   // GBK_TO_UNICODE[1865] := 16#547E;
   // GBK_TO_UNICODE[1866] := 16#85ED;
   // GBK_TO_UNICODE[1867] := 16#547F;
   // GBK_TO_UNICODE[1868] := 16#85EE;
   // GBK_TO_UNICODE[1869] := 16#5481;
   // GBK_TO_UNICODE[1870] := 16#85EF;
   // GBK_TO_UNICODE[1871] := 16#5483;
   // GBK_TO_UNICODE[1872] := 16#85F0;
   // GBK_TO_UNICODE[1873] := 16#5485;
   // GBK_TO_UNICODE[1874] := 16#85F1;
   // GBK_TO_UNICODE[1875] := 16#5487;
   // GBK_TO_UNICODE[1876] := 16#85F2;
   // GBK_TO_UNICODE[1877] := 16#5488;
   // GBK_TO_UNICODE[1878] := 16#85F3;
   // GBK_TO_UNICODE[1879] := 16#5489;
   // GBK_TO_UNICODE[1880] := 16#85F4;
   // GBK_TO_UNICODE[1881] := 16#548A;
   // GBK_TO_UNICODE[1882] := 16#85F5;
   // GBK_TO_UNICODE[1883] := 16#548D;
   // GBK_TO_UNICODE[1884] := 16#85F6;
   // GBK_TO_UNICODE[1885] := 16#5491;
   // GBK_TO_UNICODE[1886] := 16#85F7;
   // GBK_TO_UNICODE[1887] := 16#5493;
   // GBK_TO_UNICODE[1888] := 16#85F8;
   // GBK_TO_UNICODE[1889] := 16#5497;
   // GBK_TO_UNICODE[1890] := 16#85F9;
   // GBK_TO_UNICODE[1891] := 16#5498;
   // GBK_TO_UNICODE[1892] := 16#85FA;
   // GBK_TO_UNICODE[1893] := 16#549C;
   // GBK_TO_UNICODE[1894] := 16#85FB;
   // GBK_TO_UNICODE[1895] := 16#549E;
   // GBK_TO_UNICODE[1896] := 16#85FC;
   // GBK_TO_UNICODE[1897] := 16#549F;
   // GBK_TO_UNICODE[1898] := 16#85FD;
   // GBK_TO_UNICODE[1899] := 16#54A0;
   // GBK_TO_UNICODE[1900] := 16#85FE;
   // GBK_TO_UNICODE[1901] := 16#54A1;
   // GBK_TO_UNICODE[1902] := 16#8640;
   // GBK_TO_UNICODE[1903] := 16#54A2;
   // GBK_TO_UNICODE[1904] := 16#8641;
   // GBK_TO_UNICODE[1905] := 16#54A5;
   // GBK_TO_UNICODE[1906] := 16#8642;
   // GBK_TO_UNICODE[1907] := 16#54AE;
   // GBK_TO_UNICODE[1908] := 16#8643;
   // GBK_TO_UNICODE[1909] := 16#54B0;
   // GBK_TO_UNICODE[1910] := 16#8644;
   // GBK_TO_UNICODE[1911] := 16#54B2;
   // GBK_TO_UNICODE[1912] := 16#8645;
   // GBK_TO_UNICODE[1913] := 16#54B5;
   // GBK_TO_UNICODE[1914] := 16#8646;
   // GBK_TO_UNICODE[1915] := 16#54B6;
   // GBK_TO_UNICODE[1916] := 16#8647;
   // GBK_TO_UNICODE[1917] := 16#54B7;
   // GBK_TO_UNICODE[1918] := 16#8648;
   // GBK_TO_UNICODE[1919] := 16#54B9;
   // GBK_TO_UNICODE[1920] := 16#8649;
   // GBK_TO_UNICODE[1921] := 16#54BA;
   // GBK_TO_UNICODE[1922] := 16#864A;
   // GBK_TO_UNICODE[1923] := 16#54BC;
   // GBK_TO_UNICODE[1924] := 16#864B;
   // GBK_TO_UNICODE[1925] := 16#54BE;
   // GBK_TO_UNICODE[1926] := 16#864C;
   // GBK_TO_UNICODE[1927] := 16#54C3;
   // GBK_TO_UNICODE[1928] := 16#864D;
   // GBK_TO_UNICODE[1929] := 16#54C5;
   // GBK_TO_UNICODE[1930] := 16#864E;
   // GBK_TO_UNICODE[1931] := 16#54CA;
   // GBK_TO_UNICODE[1932] := 16#864F;
   // GBK_TO_UNICODE[1933] := 16#54CB;
   // GBK_TO_UNICODE[1934] := 16#8650;
   // GBK_TO_UNICODE[1935] := 16#54D6;
   // GBK_TO_UNICODE[1936] := 16#8651;
   // GBK_TO_UNICODE[1937] := 16#54D8;
   // GBK_TO_UNICODE[1938] := 16#8652;
   // GBK_TO_UNICODE[1939] := 16#54DB;
   // GBK_TO_UNICODE[1940] := 16#8653;
   // GBK_TO_UNICODE[1941] := 16#54E0;
   // GBK_TO_UNICODE[1942] := 16#8654;
   // GBK_TO_UNICODE[1943] := 16#54E1;
   // GBK_TO_UNICODE[1944] := 16#8655;
   // GBK_TO_UNICODE[1945] := 16#54E2;
   // GBK_TO_UNICODE[1946] := 16#8656;
   // GBK_TO_UNICODE[1947] := 16#54E3;
   // GBK_TO_UNICODE[1948] := 16#8657;
   // GBK_TO_UNICODE[1949] := 16#54E4;
   // GBK_TO_UNICODE[1950] := 16#8658;
   // GBK_TO_UNICODE[1951] := 16#54EB;
   // GBK_TO_UNICODE[1952] := 16#8659;
   // GBK_TO_UNICODE[1953] := 16#54EC;
   // GBK_TO_UNICODE[1954] := 16#865A;
   // GBK_TO_UNICODE[1955] := 16#54EF;
   // GBK_TO_UNICODE[1956] := 16#865B;
   // GBK_TO_UNICODE[1957] := 16#54F0;
   // GBK_TO_UNICODE[1958] := 16#865C;
   // GBK_TO_UNICODE[1959] := 16#54F1;
   // GBK_TO_UNICODE[1960] := 16#865D;
   // GBK_TO_UNICODE[1961] := 16#54F4;
   // GBK_TO_UNICODE[1962] := 16#865E;
   // GBK_TO_UNICODE[1963] := 16#54F5;
   // GBK_TO_UNICODE[1964] := 16#865F;
   // GBK_TO_UNICODE[1965] := 16#54F6;
   // GBK_TO_UNICODE[1966] := 16#8660;
   // GBK_TO_UNICODE[1967] := 16#54F7;
   // GBK_TO_UNICODE[1968] := 16#8661;
   // GBK_TO_UNICODE[1969] := 16#54F8;
   // GBK_TO_UNICODE[1970] := 16#8662;
   // GBK_TO_UNICODE[1971] := 16#54F9;
   // GBK_TO_UNICODE[1972] := 16#8663;
   // GBK_TO_UNICODE[1973] := 16#54FB;
   // GBK_TO_UNICODE[1974] := 16#8664;
   // GBK_TO_UNICODE[1975] := 16#54FE;
   // GBK_TO_UNICODE[1976] := 16#8665;
   // GBK_TO_UNICODE[1977] := 16#5500;
   // GBK_TO_UNICODE[1978] := 16#8666;
   // GBK_TO_UNICODE[1979] := 16#5502;
   // GBK_TO_UNICODE[1980] := 16#8667;
   // GBK_TO_UNICODE[1981] := 16#5503;
   // GBK_TO_UNICODE[1982] := 16#8668;
   // GBK_TO_UNICODE[1983] := 16#5504;
   // GBK_TO_UNICODE[1984] := 16#8669;
   // GBK_TO_UNICODE[1985] := 16#5505;
   // GBK_TO_UNICODE[1986] := 16#866A;
   // GBK_TO_UNICODE[1987] := 16#5508;
   // GBK_TO_UNICODE[1988] := 16#866B;
   // GBK_TO_UNICODE[1989] := 16#550A;
   // GBK_TO_UNICODE[1990] := 16#866C;
   // GBK_TO_UNICODE[1991] := 16#550B;
   // GBK_TO_UNICODE[1992] := 16#866D;
   // GBK_TO_UNICODE[1993] := 16#550C;
   // GBK_TO_UNICODE[1994] := 16#866E;
   // GBK_TO_UNICODE[1995] := 16#550D;
   // GBK_TO_UNICODE[1996] := 16#866F;
   // GBK_TO_UNICODE[1997] := 16#550E;
   // GBK_TO_UNICODE[1998] := 16#8670;
   // GBK_TO_UNICODE[1999] := 16#5512;
   // GBK_TO_UNICODE[2000] := 16#8671;
   // GBK_TO_UNICODE[2001] := 16#5513;
   // GBK_TO_UNICODE[2002] := 16#8672;
   // GBK_TO_UNICODE[2003] := 16#5515;
   // GBK_TO_UNICODE[2004] := 16#8673;
   // GBK_TO_UNICODE[2005] := 16#5516;
   // GBK_TO_UNICODE[2006] := 16#8674;
   // GBK_TO_UNICODE[2007] := 16#5517;
   // GBK_TO_UNICODE[2008] := 16#8675;
   // GBK_TO_UNICODE[2009] := 16#5518;
   // GBK_TO_UNICODE[2010] := 16#8676;
   // GBK_TO_UNICODE[2011] := 16#5519;
   // GBK_TO_UNICODE[2012] := 16#8677;
   // GBK_TO_UNICODE[2013] := 16#551A;
   // GBK_TO_UNICODE[2014] := 16#8678;
   // GBK_TO_UNICODE[2015] := 16#551C;
   // GBK_TO_UNICODE[2016] := 16#8679;
   // GBK_TO_UNICODE[2017] := 16#551D;
   // GBK_TO_UNICODE[2018] := 16#867A;
   // GBK_TO_UNICODE[2019] := 16#551E;
   // GBK_TO_UNICODE[2020] := 16#867B;
   // GBK_TO_UNICODE[2021] := 16#551F;
   // GBK_TO_UNICODE[2022] := 16#867C;
   // GBK_TO_UNICODE[2023] := 16#5521;
   // GBK_TO_UNICODE[2024] := 16#867D;
   // GBK_TO_UNICODE[2025] := 16#5525;
   // GBK_TO_UNICODE[2026] := 16#867E;
   // GBK_TO_UNICODE[2027] := 16#5526;
   // GBK_TO_UNICODE[2028] := 16#8680;
   // GBK_TO_UNICODE[2029] := 16#5528;
   // GBK_TO_UNICODE[2030] := 16#8681;
   // GBK_TO_UNICODE[2031] := 16#5529;
   // GBK_TO_UNICODE[2032] := 16#8682;
   // GBK_TO_UNICODE[2033] := 16#552B;
   // GBK_TO_UNICODE[2034] := 16#8683;
   // GBK_TO_UNICODE[2035] := 16#552D;
   // GBK_TO_UNICODE[2036] := 16#8684;
   // GBK_TO_UNICODE[2037] := 16#5532;
   // GBK_TO_UNICODE[2038] := 16#8685;
   // GBK_TO_UNICODE[2039] := 16#5534;
   // GBK_TO_UNICODE[2040] := 16#8686;
   // GBK_TO_UNICODE[2041] := 16#5535;
   // GBK_TO_UNICODE[2042] := 16#8687;
   // GBK_TO_UNICODE[2043] := 16#5536;
   // GBK_TO_UNICODE[2044] := 16#8688;
   // GBK_TO_UNICODE[2045] := 16#5538;
   // GBK_TO_UNICODE[2046] := 16#8689;
   // GBK_TO_UNICODE[2047] := 16#5539;
   // GBK_TO_UNICODE[2048] := 16#868A;
   // GBK_TO_UNICODE[2049] := 16#553A;
   // GBK_TO_UNICODE[2050] := 16#868B;
   // GBK_TO_UNICODE[2051] := 16#553B;
   // GBK_TO_UNICODE[2052] := 16#868C;
   // GBK_TO_UNICODE[2053] := 16#553D;
   // GBK_TO_UNICODE[2054] := 16#868D;
   // GBK_TO_UNICODE[2055] := 16#5540;
   // GBK_TO_UNICODE[2056] := 16#868E;
   // GBK_TO_UNICODE[2057] := 16#5542;
   // GBK_TO_UNICODE[2058] := 16#868F;
   // GBK_TO_UNICODE[2059] := 16#5545;
   // GBK_TO_UNICODE[2060] := 16#8690;
   // GBK_TO_UNICODE[2061] := 16#5547;
   // GBK_TO_UNICODE[2062] := 16#8691;
   // GBK_TO_UNICODE[2063] := 16#5548;
   // GBK_TO_UNICODE[2064] := 16#8692;
   // GBK_TO_UNICODE[2065] := 16#554B;
   // GBK_TO_UNICODE[2066] := 16#8693;
   // GBK_TO_UNICODE[2067] := 16#554C;
   // GBK_TO_UNICODE[2068] := 16#8694;
   // GBK_TO_UNICODE[2069] := 16#554D;
   // GBK_TO_UNICODE[2070] := 16#8695;
   // GBK_TO_UNICODE[2071] := 16#554E;
   // GBK_TO_UNICODE[2072] := 16#8696;
   // GBK_TO_UNICODE[2073] := 16#554F;
   // GBK_TO_UNICODE[2074] := 16#8697;
   // GBK_TO_UNICODE[2075] := 16#5551;
   // GBK_TO_UNICODE[2076] := 16#8698;
   // GBK_TO_UNICODE[2077] := 16#5552;
   // GBK_TO_UNICODE[2078] := 16#8699;
   // GBK_TO_UNICODE[2079] := 16#5553;
   // GBK_TO_UNICODE[2080] := 16#869A;
   // GBK_TO_UNICODE[2081] := 16#5554;
   // GBK_TO_UNICODE[2082] := 16#869B;
   // GBK_TO_UNICODE[2083] := 16#5557;
   // GBK_TO_UNICODE[2084] := 16#869C;
   // GBK_TO_UNICODE[2085] := 16#5558;
   // GBK_TO_UNICODE[2086] := 16#869D;
   // GBK_TO_UNICODE[2087] := 16#5559;
   // GBK_TO_UNICODE[2088] := 16#869E;
   // GBK_TO_UNICODE[2089] := 16#555A;
   // GBK_TO_UNICODE[2090] := 16#869F;
   // GBK_TO_UNICODE[2091] := 16#555B;
   // GBK_TO_UNICODE[2092] := 16#86A0;
   // GBK_TO_UNICODE[2093] := 16#555D;
   // GBK_TO_UNICODE[2094] := 16#86A1;
   // GBK_TO_UNICODE[2095] := 16#555E;
   // GBK_TO_UNICODE[2096] := 16#86A2;
   // GBK_TO_UNICODE[2097] := 16#555F;
   // GBK_TO_UNICODE[2098] := 16#86A3;
   // GBK_TO_UNICODE[2099] := 16#5560;
   // GBK_TO_UNICODE[2100] := 16#86A4;
   // GBK_TO_UNICODE[2101] := 16#5562;
   // GBK_TO_UNICODE[2102] := 16#86A5;
   // GBK_TO_UNICODE[2103] := 16#5563;
   // GBK_TO_UNICODE[2104] := 16#86A6;
   // GBK_TO_UNICODE[2105] := 16#5568;
   // GBK_TO_UNICODE[2106] := 16#86A7;
   // GBK_TO_UNICODE[2107] := 16#5569;
   // GBK_TO_UNICODE[2108] := 16#86A8;
   // GBK_TO_UNICODE[2109] := 16#556B;
   // GBK_TO_UNICODE[2110] := 16#86A9;
   // GBK_TO_UNICODE[2111] := 16#556F;
   // GBK_TO_UNICODE[2112] := 16#86AA;
   // GBK_TO_UNICODE[2113] := 16#5570;
   // GBK_TO_UNICODE[2114] := 16#86AB;
   // GBK_TO_UNICODE[2115] := 16#5571;
   // GBK_TO_UNICODE[2116] := 16#86AC;
   // GBK_TO_UNICODE[2117] := 16#5572;
   // GBK_TO_UNICODE[2118] := 16#86AD;
   // GBK_TO_UNICODE[2119] := 16#5573;
   // GBK_TO_UNICODE[2120] := 16#86AE;
   // GBK_TO_UNICODE[2121] := 16#5574;
   // GBK_TO_UNICODE[2122] := 16#86AF;
   // GBK_TO_UNICODE[2123] := 16#5579;
   // GBK_TO_UNICODE[2124] := 16#86B0;
   // GBK_TO_UNICODE[2125] := 16#557A;
   // GBK_TO_UNICODE[2126] := 16#86B1;
   // GBK_TO_UNICODE[2127] := 16#557D;
   // GBK_TO_UNICODE[2128] := 16#86B2;
   // GBK_TO_UNICODE[2129] := 16#557F;
   // GBK_TO_UNICODE[2130] := 16#86B3;
   // GBK_TO_UNICODE[2131] := 16#5585;
   // GBK_TO_UNICODE[2132] := 16#86B4;
   // GBK_TO_UNICODE[2133] := 16#5586;
   // GBK_TO_UNICODE[2134] := 16#86B5;
   // GBK_TO_UNICODE[2135] := 16#558C;
   // GBK_TO_UNICODE[2136] := 16#86B6;
   // GBK_TO_UNICODE[2137] := 16#558D;
   // GBK_TO_UNICODE[2138] := 16#86B7;
   // GBK_TO_UNICODE[2139] := 16#558E;
   // GBK_TO_UNICODE[2140] := 16#86B8;
   // GBK_TO_UNICODE[2141] := 16#5590;
   // GBK_TO_UNICODE[2142] := 16#86B9;
   // GBK_TO_UNICODE[2143] := 16#5592;
   // GBK_TO_UNICODE[2144] := 16#86BA;
   // GBK_TO_UNICODE[2145] := 16#5593;
   // GBK_TO_UNICODE[2146] := 16#86BB;
   // GBK_TO_UNICODE[2147] := 16#5595;
   // GBK_TO_UNICODE[2148] := 16#86BC;
   // GBK_TO_UNICODE[2149] := 16#5596;
   // GBK_TO_UNICODE[2150] := 16#86BD;
   // GBK_TO_UNICODE[2151] := 16#5597;
   // GBK_TO_UNICODE[2152] := 16#86BE;
   // GBK_TO_UNICODE[2153] := 16#559A;
   // GBK_TO_UNICODE[2154] := 16#86BF;
   // GBK_TO_UNICODE[2155] := 16#559B;
   // GBK_TO_UNICODE[2156] := 16#86C0;
   // GBK_TO_UNICODE[2157] := 16#559E;
   // GBK_TO_UNICODE[2158] := 16#86C1;
   // GBK_TO_UNICODE[2159] := 16#55A0;
   // GBK_TO_UNICODE[2160] := 16#86C2;
   // GBK_TO_UNICODE[2161] := 16#55A1;
   // GBK_TO_UNICODE[2162] := 16#86C3;
   // GBK_TO_UNICODE[2163] := 16#55A2;
   // GBK_TO_UNICODE[2164] := 16#86C4;
   // GBK_TO_UNICODE[2165] := 16#55A3;
   // GBK_TO_UNICODE[2166] := 16#86C5;
   // GBK_TO_UNICODE[2167] := 16#55A4;
   // GBK_TO_UNICODE[2168] := 16#86C6;
   // GBK_TO_UNICODE[2169] := 16#55A5;
   // GBK_TO_UNICODE[2170] := 16#86C7;
   // GBK_TO_UNICODE[2171] := 16#55A6;
   // GBK_TO_UNICODE[2172] := 16#86C8;
   // GBK_TO_UNICODE[2173] := 16#55A8;
   // GBK_TO_UNICODE[2174] := 16#86C9;
   // GBK_TO_UNICODE[2175] := 16#55A9;
   // GBK_TO_UNICODE[2176] := 16#86CA;
   // GBK_TO_UNICODE[2177] := 16#55AA;
   // GBK_TO_UNICODE[2178] := 16#86CB;
   // GBK_TO_UNICODE[2179] := 16#55AB;
   // GBK_TO_UNICODE[2180] := 16#86CC;
   // GBK_TO_UNICODE[2181] := 16#55AC;
   // GBK_TO_UNICODE[2182] := 16#86CD;
   // GBK_TO_UNICODE[2183] := 16#55AD;
   // GBK_TO_UNICODE[2184] := 16#86CE;
   // GBK_TO_UNICODE[2185] := 16#55AE;
   // GBK_TO_UNICODE[2186] := 16#86CF;
   // GBK_TO_UNICODE[2187] := 16#55AF;
   // GBK_TO_UNICODE[2188] := 16#86D0;
   // GBK_TO_UNICODE[2189] := 16#55B0;
   // GBK_TO_UNICODE[2190] := 16#86D1;
   // GBK_TO_UNICODE[2191] := 16#55B2;
   // GBK_TO_UNICODE[2192] := 16#86D2;
   // GBK_TO_UNICODE[2193] := 16#55B4;
   // GBK_TO_UNICODE[2194] := 16#86D3;
   // GBK_TO_UNICODE[2195] := 16#55B6;
   // GBK_TO_UNICODE[2196] := 16#86D4;
   // GBK_TO_UNICODE[2197] := 16#55B8;
   // GBK_TO_UNICODE[2198] := 16#86D5;
   // GBK_TO_UNICODE[2199] := 16#55BA;
   // GBK_TO_UNICODE[2200] := 16#86D6;
   // GBK_TO_UNICODE[2201] := 16#55BC;
   // GBK_TO_UNICODE[2202] := 16#86D7;
   // GBK_TO_UNICODE[2203] := 16#55BF;
   // GBK_TO_UNICODE[2204] := 16#86D8;
   // GBK_TO_UNICODE[2205] := 16#55C0;
   // GBK_TO_UNICODE[2206] := 16#86D9;
   // GBK_TO_UNICODE[2207] := 16#55C1;
   // GBK_TO_UNICODE[2208] := 16#86DA;
   // GBK_TO_UNICODE[2209] := 16#55C2;
   // GBK_TO_UNICODE[2210] := 16#86DB;
   // GBK_TO_UNICODE[2211] := 16#55C3;
   // GBK_TO_UNICODE[2212] := 16#86DC;
   // GBK_TO_UNICODE[2213] := 16#55C6;
   // GBK_TO_UNICODE[2214] := 16#86DD;
   // GBK_TO_UNICODE[2215] := 16#55C7;
   // GBK_TO_UNICODE[2216] := 16#86DE;
   // GBK_TO_UNICODE[2217] := 16#55C8;
   // GBK_TO_UNICODE[2218] := 16#86DF;
   // GBK_TO_UNICODE[2219] := 16#55CA;
   // GBK_TO_UNICODE[2220] := 16#86E0;
   // GBK_TO_UNICODE[2221] := 16#55CB;
   // GBK_TO_UNICODE[2222] := 16#86E1;
   // GBK_TO_UNICODE[2223] := 16#55CE;
   // GBK_TO_UNICODE[2224] := 16#86E2;
   // GBK_TO_UNICODE[2225] := 16#55CF;
   // GBK_TO_UNICODE[2226] := 16#86E3;
   // GBK_TO_UNICODE[2227] := 16#55D0;
   // GBK_TO_UNICODE[2228] := 16#86E4;
   // GBK_TO_UNICODE[2229] := 16#55D5;
   // GBK_TO_UNICODE[2230] := 16#86E5;
   // GBK_TO_UNICODE[2231] := 16#55D7;
   // GBK_TO_UNICODE[2232] := 16#86E6;
   // GBK_TO_UNICODE[2233] := 16#55D8;
   // GBK_TO_UNICODE[2234] := 16#86E7;
   // GBK_TO_UNICODE[2235] := 16#55D9;
   // GBK_TO_UNICODE[2236] := 16#86E8;
   // GBK_TO_UNICODE[2237] := 16#55DA;
   // GBK_TO_UNICODE[2238] := 16#86E9;
   // GBK_TO_UNICODE[2239] := 16#55DB;
   // GBK_TO_UNICODE[2240] := 16#86EA;
   // GBK_TO_UNICODE[2241] := 16#55DE;
   // GBK_TO_UNICODE[2242] := 16#86EB;
   // GBK_TO_UNICODE[2243] := 16#55E0;
   // GBK_TO_UNICODE[2244] := 16#86EC;
   // GBK_TO_UNICODE[2245] := 16#55E2;
   // GBK_TO_UNICODE[2246] := 16#86ED;
   // GBK_TO_UNICODE[2247] := 16#55E7;
   // GBK_TO_UNICODE[2248] := 16#86EE;
   // GBK_TO_UNICODE[2249] := 16#55E9;
   // GBK_TO_UNICODE[2250] := 16#86EF;
   // GBK_TO_UNICODE[2251] := 16#55ED;
   // GBK_TO_UNICODE[2252] := 16#86F0;
   // GBK_TO_UNICODE[2253] := 16#55EE;
   // GBK_TO_UNICODE[2254] := 16#86F1;
   // GBK_TO_UNICODE[2255] := 16#55F0;
   // GBK_TO_UNICODE[2256] := 16#86F2;
   // GBK_TO_UNICODE[2257] := 16#55F1;
   // GBK_TO_UNICODE[2258] := 16#86F3;
   // GBK_TO_UNICODE[2259] := 16#55F4;
   // GBK_TO_UNICODE[2260] := 16#86F4;
   // GBK_TO_UNICODE[2261] := 16#55F6;
   // GBK_TO_UNICODE[2262] := 16#86F5;
   // GBK_TO_UNICODE[2263] := 16#55F8;
   // GBK_TO_UNICODE[2264] := 16#86F6;
   // GBK_TO_UNICODE[2265] := 16#55F9;
   // GBK_TO_UNICODE[2266] := 16#86F7;
   // GBK_TO_UNICODE[2267] := 16#55FA;
   // GBK_TO_UNICODE[2268] := 16#86F8;
   // GBK_TO_UNICODE[2269] := 16#55FB;
   // GBK_TO_UNICODE[2270] := 16#86F9;
   // GBK_TO_UNICODE[2271] := 16#55FC;
   // GBK_TO_UNICODE[2272] := 16#86FA;
   // GBK_TO_UNICODE[2273] := 16#55FF;
   // GBK_TO_UNICODE[2274] := 16#86FB;
   // GBK_TO_UNICODE[2275] := 16#5602;
   // GBK_TO_UNICODE[2276] := 16#86FC;
   // GBK_TO_UNICODE[2277] := 16#5603;
   // GBK_TO_UNICODE[2278] := 16#86FD;
   // GBK_TO_UNICODE[2279] := 16#5604;
   // GBK_TO_UNICODE[2280] := 16#86FE;
   // GBK_TO_UNICODE[2281] := 16#5605;
   // GBK_TO_UNICODE[2282] := 16#8740;
   // GBK_TO_UNICODE[2283] := 16#5606;
   // GBK_TO_UNICODE[2284] := 16#8741;
   // GBK_TO_UNICODE[2285] := 16#5607;
   // GBK_TO_UNICODE[2286] := 16#8742;
   // GBK_TO_UNICODE[2287] := 16#560A;
   // GBK_TO_UNICODE[2288] := 16#8743;
   // GBK_TO_UNICODE[2289] := 16#560B;
   // GBK_TO_UNICODE[2290] := 16#8744;
   // GBK_TO_UNICODE[2291] := 16#560D;
   // GBK_TO_UNICODE[2292] := 16#8745;
   // GBK_TO_UNICODE[2293] := 16#5610;
   // GBK_TO_UNICODE[2294] := 16#8746;
   // GBK_TO_UNICODE[2295] := 16#5611;
   // GBK_TO_UNICODE[2296] := 16#8747;
   // GBK_TO_UNICODE[2297] := 16#5612;
   // GBK_TO_UNICODE[2298] := 16#8748;
   // GBK_TO_UNICODE[2299] := 16#5613;
   // GBK_TO_UNICODE[2300] := 16#8749;
   // GBK_TO_UNICODE[2301] := 16#5614;
   // GBK_TO_UNICODE[2302] := 16#874A;
   // GBK_TO_UNICODE[2303] := 16#5615;
   // GBK_TO_UNICODE[2304] := 16#874B;
   // GBK_TO_UNICODE[2305] := 16#5616;
   // GBK_TO_UNICODE[2306] := 16#874C;
   // GBK_TO_UNICODE[2307] := 16#5617;
   // GBK_TO_UNICODE[2308] := 16#874D;
   // GBK_TO_UNICODE[2309] := 16#5619;
   // GBK_TO_UNICODE[2310] := 16#874E;
   // GBK_TO_UNICODE[2311] := 16#561A;
   // GBK_TO_UNICODE[2312] := 16#874F;
   // GBK_TO_UNICODE[2313] := 16#561C;
   // GBK_TO_UNICODE[2314] := 16#8750;
   // GBK_TO_UNICODE[2315] := 16#561D;
   // GBK_TO_UNICODE[2316] := 16#8751;
   // GBK_TO_UNICODE[2317] := 16#5620;
   // GBK_TO_UNICODE[2318] := 16#8752;
   // GBK_TO_UNICODE[2319] := 16#5621;
   // GBK_TO_UNICODE[2320] := 16#8753;
   // GBK_TO_UNICODE[2321] := 16#5622;
   // GBK_TO_UNICODE[2322] := 16#8754;
   // GBK_TO_UNICODE[2323] := 16#5625;
   // GBK_TO_UNICODE[2324] := 16#8755;
   // GBK_TO_UNICODE[2325] := 16#5626;
   // GBK_TO_UNICODE[2326] := 16#8756;
   // GBK_TO_UNICODE[2327] := 16#5628;
   // GBK_TO_UNICODE[2328] := 16#8757;
   // GBK_TO_UNICODE[2329] := 16#5629;
   // GBK_TO_UNICODE[2330] := 16#8758;
   // GBK_TO_UNICODE[2331] := 16#562A;
   // GBK_TO_UNICODE[2332] := 16#8759;
   // GBK_TO_UNICODE[2333] := 16#562B;
   // GBK_TO_UNICODE[2334] := 16#875A;
   // GBK_TO_UNICODE[2335] := 16#562E;
   // GBK_TO_UNICODE[2336] := 16#875B;
   // GBK_TO_UNICODE[2337] := 16#562F;
   // GBK_TO_UNICODE[2338] := 16#875C;
   // GBK_TO_UNICODE[2339] := 16#5630;
   // GBK_TO_UNICODE[2340] := 16#875D;
   // GBK_TO_UNICODE[2341] := 16#5633;
   // GBK_TO_UNICODE[2342] := 16#875E;
   // GBK_TO_UNICODE[2343] := 16#5635;
   // GBK_TO_UNICODE[2344] := 16#875F;
   // GBK_TO_UNICODE[2345] := 16#5637;
   // GBK_TO_UNICODE[2346] := 16#8760;
   // GBK_TO_UNICODE[2347] := 16#5638;
   // GBK_TO_UNICODE[2348] := 16#8761;
   // GBK_TO_UNICODE[2349] := 16#563A;
   // GBK_TO_UNICODE[2350] := 16#8762;
   // GBK_TO_UNICODE[2351] := 16#563C;
   // GBK_TO_UNICODE[2352] := 16#8763;
   // GBK_TO_UNICODE[2353] := 16#563D;
   // GBK_TO_UNICODE[2354] := 16#8764;
   // GBK_TO_UNICODE[2355] := 16#563E;
   // GBK_TO_UNICODE[2356] := 16#8765;
   // GBK_TO_UNICODE[2357] := 16#5640;
   // GBK_TO_UNICODE[2358] := 16#8766;
   // GBK_TO_UNICODE[2359] := 16#5641;
   // GBK_TO_UNICODE[2360] := 16#8767;
   // GBK_TO_UNICODE[2361] := 16#5642;
   // GBK_TO_UNICODE[2362] := 16#8768;
   // GBK_TO_UNICODE[2363] := 16#5643;
   // GBK_TO_UNICODE[2364] := 16#8769;
   // GBK_TO_UNICODE[2365] := 16#5644;
   // GBK_TO_UNICODE[2366] := 16#876A;
   // GBK_TO_UNICODE[2367] := 16#5645;
   // GBK_TO_UNICODE[2368] := 16#876B;
   // GBK_TO_UNICODE[2369] := 16#5646;
   // GBK_TO_UNICODE[2370] := 16#876C;
   // GBK_TO_UNICODE[2371] := 16#5647;
   // GBK_TO_UNICODE[2372] := 16#876D;
   // GBK_TO_UNICODE[2373] := 16#5648;
   // GBK_TO_UNICODE[2374] := 16#876E;
   // GBK_TO_UNICODE[2375] := 16#5649;
   // GBK_TO_UNICODE[2376] := 16#876F;
   // GBK_TO_UNICODE[2377] := 16#564A;
   // GBK_TO_UNICODE[2378] := 16#8770;
   // GBK_TO_UNICODE[2379] := 16#564B;
   // GBK_TO_UNICODE[2380] := 16#8771;
   // GBK_TO_UNICODE[2381] := 16#564F;
   // GBK_TO_UNICODE[2382] := 16#8772;
   // GBK_TO_UNICODE[2383] := 16#5650;
   // GBK_TO_UNICODE[2384] := 16#8773;
   // GBK_TO_UNICODE[2385] := 16#5651;
   // GBK_TO_UNICODE[2386] := 16#8774;
   // GBK_TO_UNICODE[2387] := 16#5652;
   // GBK_TO_UNICODE[2388] := 16#8775;
   // GBK_TO_UNICODE[2389] := 16#5653;
   // GBK_TO_UNICODE[2390] := 16#8776;
   // GBK_TO_UNICODE[2391] := 16#5655;
   // GBK_TO_UNICODE[2392] := 16#8777;
   // GBK_TO_UNICODE[2393] := 16#5656;
   // GBK_TO_UNICODE[2394] := 16#8778;
   // GBK_TO_UNICODE[2395] := 16#565A;
   // GBK_TO_UNICODE[2396] := 16#8779;
   // GBK_TO_UNICODE[2397] := 16#565B;
   // GBK_TO_UNICODE[2398] := 16#877A;
   // GBK_TO_UNICODE[2399] := 16#565D;
   // GBK_TO_UNICODE[2400] := 16#877B;
   // GBK_TO_UNICODE[2401] := 16#565E;
   // GBK_TO_UNICODE[2402] := 16#877C;
   // GBK_TO_UNICODE[2403] := 16#565F;
   // GBK_TO_UNICODE[2404] := 16#877D;
   // GBK_TO_UNICODE[2405] := 16#5660;
   // GBK_TO_UNICODE[2406] := 16#877E;
   // GBK_TO_UNICODE[2407] := 16#5661;
   // GBK_TO_UNICODE[2408] := 16#8780;
   // GBK_TO_UNICODE[2409] := 16#5663;
   // GBK_TO_UNICODE[2410] := 16#8781;
   // GBK_TO_UNICODE[2411] := 16#5665;
   // GBK_TO_UNICODE[2412] := 16#8782;
   // GBK_TO_UNICODE[2413] := 16#5666;
   // GBK_TO_UNICODE[2414] := 16#8783;
   // GBK_TO_UNICODE[2415] := 16#5667;
   // GBK_TO_UNICODE[2416] := 16#8784;
   // GBK_TO_UNICODE[2417] := 16#566D;
   // GBK_TO_UNICODE[2418] := 16#8785;
   // GBK_TO_UNICODE[2419] := 16#566E;
   // GBK_TO_UNICODE[2420] := 16#8786;
   // GBK_TO_UNICODE[2421] := 16#566F;
   // GBK_TO_UNICODE[2422] := 16#8787;
   // GBK_TO_UNICODE[2423] := 16#5670;
   // GBK_TO_UNICODE[2424] := 16#8788;
   // GBK_TO_UNICODE[2425] := 16#5672;
   // GBK_TO_UNICODE[2426] := 16#8789;
   // GBK_TO_UNICODE[2427] := 16#5673;
   // GBK_TO_UNICODE[2428] := 16#878A;
   // GBK_TO_UNICODE[2429] := 16#5674;
   // GBK_TO_UNICODE[2430] := 16#878B;
   // GBK_TO_UNICODE[2431] := 16#5675;
   // GBK_TO_UNICODE[2432] := 16#878C;
   // GBK_TO_UNICODE[2433] := 16#5677;
   // GBK_TO_UNICODE[2434] := 16#878D;
   // GBK_TO_UNICODE[2435] := 16#5678;
   // GBK_TO_UNICODE[2436] := 16#878E;
   // GBK_TO_UNICODE[2437] := 16#5679;
   // GBK_TO_UNICODE[2438] := 16#878F;
   // GBK_TO_UNICODE[2439] := 16#567A;
   // GBK_TO_UNICODE[2440] := 16#8790;
   // GBK_TO_UNICODE[2441] := 16#567D;
   // GBK_TO_UNICODE[2442] := 16#8791;
   // GBK_TO_UNICODE[2443] := 16#567E;
   // GBK_TO_UNICODE[2444] := 16#8792;
   // GBK_TO_UNICODE[2445] := 16#567F;
   // GBK_TO_UNICODE[2446] := 16#8793;
   // GBK_TO_UNICODE[2447] := 16#5680;
   // GBK_TO_UNICODE[2448] := 16#8794;
   // GBK_TO_UNICODE[2449] := 16#5681;
   // GBK_TO_UNICODE[2450] := 16#8795;
   // GBK_TO_UNICODE[2451] := 16#5682;
   // GBK_TO_UNICODE[2452] := 16#8796;
   // GBK_TO_UNICODE[2453] := 16#5683;
   // GBK_TO_UNICODE[2454] := 16#8797;
   // GBK_TO_UNICODE[2455] := 16#5684;
   // GBK_TO_UNICODE[2456] := 16#8798;
   // GBK_TO_UNICODE[2457] := 16#5687;
   // GBK_TO_UNICODE[2458] := 16#8799;
   // GBK_TO_UNICODE[2459] := 16#5688;
   // GBK_TO_UNICODE[2460] := 16#879A;
   // GBK_TO_UNICODE[2461] := 16#5689;
   // GBK_TO_UNICODE[2462] := 16#879B;
   // GBK_TO_UNICODE[2463] := 16#568A;
   // GBK_TO_UNICODE[2464] := 16#879C;
   // GBK_TO_UNICODE[2465] := 16#568B;
   // GBK_TO_UNICODE[2466] := 16#879D;
   // GBK_TO_UNICODE[2467] := 16#568C;
   // GBK_TO_UNICODE[2468] := 16#879E;
   // GBK_TO_UNICODE[2469] := 16#568D;
   // GBK_TO_UNICODE[2470] := 16#879F;
   // GBK_TO_UNICODE[2471] := 16#5690;
   // GBK_TO_UNICODE[2472] := 16#87A0;
   // GBK_TO_UNICODE[2473] := 16#5691;
   // GBK_TO_UNICODE[2474] := 16#87A1;
   // GBK_TO_UNICODE[2475] := 16#5692;
   // GBK_TO_UNICODE[2476] := 16#87A2;
   // GBK_TO_UNICODE[2477] := 16#5694;
   // GBK_TO_UNICODE[2478] := 16#87A3;
   // GBK_TO_UNICODE[2479] := 16#5695;
   // GBK_TO_UNICODE[2480] := 16#87A4;
   // GBK_TO_UNICODE[2481] := 16#5696;
   // GBK_TO_UNICODE[2482] := 16#87A5;
   // GBK_TO_UNICODE[2483] := 16#5697;
   // GBK_TO_UNICODE[2484] := 16#87A6;
   // GBK_TO_UNICODE[2485] := 16#5698;
   // GBK_TO_UNICODE[2486] := 16#87A7;
   // GBK_TO_UNICODE[2487] := 16#5699;
   // GBK_TO_UNICODE[2488] := 16#87A8;
   // GBK_TO_UNICODE[2489] := 16#569A;
   // GBK_TO_UNICODE[2490] := 16#87A9;
   // GBK_TO_UNICODE[2491] := 16#569B;
   // GBK_TO_UNICODE[2492] := 16#87AA;
   // GBK_TO_UNICODE[2493] := 16#569C;
   // GBK_TO_UNICODE[2494] := 16#87AB;
   // GBK_TO_UNICODE[2495] := 16#569D;
   // GBK_TO_UNICODE[2496] := 16#87AC;
   // GBK_TO_UNICODE[2497] := 16#569E;
   // GBK_TO_UNICODE[2498] := 16#87AD;
   // GBK_TO_UNICODE[2499] := 16#569F;
   // GBK_TO_UNICODE[2500] := 16#87AE;
   // GBK_TO_UNICODE[2501] := 16#56A0;
   // GBK_TO_UNICODE[2502] := 16#87AF;
   // GBK_TO_UNICODE[2503] := 16#56A1;
   // GBK_TO_UNICODE[2504] := 16#87B0;
   // GBK_TO_UNICODE[2505] := 16#56A2;
   // GBK_TO_UNICODE[2506] := 16#87B1;
   // GBK_TO_UNICODE[2507] := 16#56A4;
   // GBK_TO_UNICODE[2508] := 16#87B2;
   // GBK_TO_UNICODE[2509] := 16#56A5;
   // GBK_TO_UNICODE[2510] := 16#87B3;
   // GBK_TO_UNICODE[2511] := 16#56A6;
   // GBK_TO_UNICODE[2512] := 16#87B4;
   // GBK_TO_UNICODE[2513] := 16#56A7;
   // GBK_TO_UNICODE[2514] := 16#87B5;
   // GBK_TO_UNICODE[2515] := 16#56A8;
   // GBK_TO_UNICODE[2516] := 16#87B6;
   // GBK_TO_UNICODE[2517] := 16#56A9;
   // GBK_TO_UNICODE[2518] := 16#87B7;
   // GBK_TO_UNICODE[2519] := 16#56AA;
   // GBK_TO_UNICODE[2520] := 16#87B8;
   // GBK_TO_UNICODE[2521] := 16#56AB;
   // GBK_TO_UNICODE[2522] := 16#87B9;
   // GBK_TO_UNICODE[2523] := 16#56AC;
   // GBK_TO_UNICODE[2524] := 16#87BA;
   // GBK_TO_UNICODE[2525] := 16#56AD;
   // GBK_TO_UNICODE[2526] := 16#87BB;
   // GBK_TO_UNICODE[2527] := 16#56AE;
   // GBK_TO_UNICODE[2528] := 16#87BC;
   // GBK_TO_UNICODE[2529] := 16#56B0;
   // GBK_TO_UNICODE[2530] := 16#87BD;
   // GBK_TO_UNICODE[2531] := 16#56B1;
   // GBK_TO_UNICODE[2532] := 16#87BE;
   // GBK_TO_UNICODE[2533] := 16#56B2;
   // GBK_TO_UNICODE[2534] := 16#87BF;
   // GBK_TO_UNICODE[2535] := 16#56B3;
   // GBK_TO_UNICODE[2536] := 16#87C0;
   // GBK_TO_UNICODE[2537] := 16#56B4;
   // GBK_TO_UNICODE[2538] := 16#87C1;
   // GBK_TO_UNICODE[2539] := 16#56B5;
   // GBK_TO_UNICODE[2540] := 16#87C2;
   // GBK_TO_UNICODE[2541] := 16#56B6;
   // GBK_TO_UNICODE[2542] := 16#87C3;
   // GBK_TO_UNICODE[2543] := 16#56B8;
   // GBK_TO_UNICODE[2544] := 16#87C4;
   // GBK_TO_UNICODE[2545] := 16#56B9;
   // GBK_TO_UNICODE[2546] := 16#87C5;
   // GBK_TO_UNICODE[2547] := 16#56BA;
   // GBK_TO_UNICODE[2548] := 16#87C6;
   // GBK_TO_UNICODE[2549] := 16#56BB;
   // GBK_TO_UNICODE[2550] := 16#87C7;
   // GBK_TO_UNICODE[2551] := 16#56BD;
   // GBK_TO_UNICODE[2552] := 16#87C8;
   // GBK_TO_UNICODE[2553] := 16#56BE;
   // GBK_TO_UNICODE[2554] := 16#87C9;
   // GBK_TO_UNICODE[2555] := 16#56BF;
   // GBK_TO_UNICODE[2556] := 16#87CA;
   // GBK_TO_UNICODE[2557] := 16#56C0;
   // GBK_TO_UNICODE[2558] := 16#87CB;
   // GBK_TO_UNICODE[2559] := 16#56C1;
   // GBK_TO_UNICODE[2560] := 16#87CC;
   // GBK_TO_UNICODE[2561] := 16#56C2;
   // GBK_TO_UNICODE[2562] := 16#87CD;
   // GBK_TO_UNICODE[2563] := 16#56C3;
   // GBK_TO_UNICODE[2564] := 16#87CE;
   // GBK_TO_UNICODE[2565] := 16#56C4;
   // GBK_TO_UNICODE[2566] := 16#87CF;
   // GBK_TO_UNICODE[2567] := 16#56C5;
   // GBK_TO_UNICODE[2568] := 16#87D0;
   // GBK_TO_UNICODE[2569] := 16#56C6;
   // GBK_TO_UNICODE[2570] := 16#87D1;
   // GBK_TO_UNICODE[2571] := 16#56C7;
   // GBK_TO_UNICODE[2572] := 16#87D2;
   // GBK_TO_UNICODE[2573] := 16#56C8;
   // GBK_TO_UNICODE[2574] := 16#87D3;
   // GBK_TO_UNICODE[2575] := 16#56C9;
   // GBK_TO_UNICODE[2576] := 16#87D4;
   // GBK_TO_UNICODE[2577] := 16#56CB;
   // GBK_TO_UNICODE[2578] := 16#87D5;
   // GBK_TO_UNICODE[2579] := 16#56CC;
   // GBK_TO_UNICODE[2580] := 16#87D6;
   // GBK_TO_UNICODE[2581] := 16#56CD;
   // GBK_TO_UNICODE[2582] := 16#87D7;
   // GBK_TO_UNICODE[2583] := 16#56CE;
   // GBK_TO_UNICODE[2584] := 16#87D8;
   // GBK_TO_UNICODE[2585] := 16#56CF;
   // GBK_TO_UNICODE[2586] := 16#87D9;
   // GBK_TO_UNICODE[2587] := 16#56D0;
   // GBK_TO_UNICODE[2588] := 16#87DA;
   // GBK_TO_UNICODE[2589] := 16#56D1;
   // GBK_TO_UNICODE[2590] := 16#87DB;
   // GBK_TO_UNICODE[2591] := 16#56D2;
   // GBK_TO_UNICODE[2592] := 16#87DC;
   // GBK_TO_UNICODE[2593] := 16#56D3;
   // GBK_TO_UNICODE[2594] := 16#87DD;
   // GBK_TO_UNICODE[2595] := 16#56D5;
   // GBK_TO_UNICODE[2596] := 16#87DE;
   // GBK_TO_UNICODE[2597] := 16#56D6;
   // GBK_TO_UNICODE[2598] := 16#87DF;
   // GBK_TO_UNICODE[2599] := 16#56D8;
   // GBK_TO_UNICODE[2600] := 16#87E0;
   // GBK_TO_UNICODE[2601] := 16#56D9;
   // GBK_TO_UNICODE[2602] := 16#87E1;
   // GBK_TO_UNICODE[2603] := 16#56DC;
   // GBK_TO_UNICODE[2604] := 16#87E2;
   // GBK_TO_UNICODE[2605] := 16#56E3;
   // GBK_TO_UNICODE[2606] := 16#87E3;
   // GBK_TO_UNICODE[2607] := 16#56E5;
   // GBK_TO_UNICODE[2608] := 16#87E4;
   // GBK_TO_UNICODE[2609] := 16#56E6;
   // GBK_TO_UNICODE[2610] := 16#87E5;
   // GBK_TO_UNICODE[2611] := 16#56E7;
   // GBK_TO_UNICODE[2612] := 16#87E6;
   // GBK_TO_UNICODE[2613] := 16#56E8;
   // GBK_TO_UNICODE[2614] := 16#87E7;
   // GBK_TO_UNICODE[2615] := 16#56E9;
   // GBK_TO_UNICODE[2616] := 16#87E8;
   // GBK_TO_UNICODE[2617] := 16#56EA;
   // GBK_TO_UNICODE[2618] := 16#87E9;
   // GBK_TO_UNICODE[2619] := 16#56EC;
   // GBK_TO_UNICODE[2620] := 16#87EA;
   // GBK_TO_UNICODE[2621] := 16#56EE;
   // GBK_TO_UNICODE[2622] := 16#87EB;
   // GBK_TO_UNICODE[2623] := 16#56EF;
   // GBK_TO_UNICODE[2624] := 16#87EC;
   // GBK_TO_UNICODE[2625] := 16#56F2;
   // GBK_TO_UNICODE[2626] := 16#87ED;
   // GBK_TO_UNICODE[2627] := 16#56F3;
   // GBK_TO_UNICODE[2628] := 16#87EE;
   // GBK_TO_UNICODE[2629] := 16#56F6;
   // GBK_TO_UNICODE[2630] := 16#87EF;
   // GBK_TO_UNICODE[2631] := 16#56F7;
   // GBK_TO_UNICODE[2632] := 16#87F0;
   // GBK_TO_UNICODE[2633] := 16#56F8;
   // GBK_TO_UNICODE[2634] := 16#87F1;
   // GBK_TO_UNICODE[2635] := 16#56FB;
   // GBK_TO_UNICODE[2636] := 16#87F2;
   // GBK_TO_UNICODE[2637] := 16#56FC;
   // GBK_TO_UNICODE[2638] := 16#87F3;
   // GBK_TO_UNICODE[2639] := 16#5700;
   // GBK_TO_UNICODE[2640] := 16#87F4;
   // GBK_TO_UNICODE[2641] := 16#5701;
   // GBK_TO_UNICODE[2642] := 16#87F5;
   // GBK_TO_UNICODE[2643] := 16#5702;
   // GBK_TO_UNICODE[2644] := 16#87F6;
   // GBK_TO_UNICODE[2645] := 16#5705;
   // GBK_TO_UNICODE[2646] := 16#87F7;
   // GBK_TO_UNICODE[2647] := 16#5707;
   // GBK_TO_UNICODE[2648] := 16#87F8;
   // GBK_TO_UNICODE[2649] := 16#570B;
   // GBK_TO_UNICODE[2650] := 16#87F9;
   // GBK_TO_UNICODE[2651] := 16#570C;
   // GBK_TO_UNICODE[2652] := 16#87FA;
   // GBK_TO_UNICODE[2653] := 16#570D;
   // GBK_TO_UNICODE[2654] := 16#87FB;
   // GBK_TO_UNICODE[2655] := 16#570E;
   // GBK_TO_UNICODE[2656] := 16#87FC;
   // GBK_TO_UNICODE[2657] := 16#570F;
   // GBK_TO_UNICODE[2658] := 16#87FD;
   // GBK_TO_UNICODE[2659] := 16#5710;
   // GBK_TO_UNICODE[2660] := 16#87FE;
   // GBK_TO_UNICODE[2661] := 16#5711;
   // GBK_TO_UNICODE[2662] := 16#8840;
   // GBK_TO_UNICODE[2663] := 16#5712;
   // GBK_TO_UNICODE[2664] := 16#8841;
   // GBK_TO_UNICODE[2665] := 16#5713;
   // GBK_TO_UNICODE[2666] := 16#8842;
   // GBK_TO_UNICODE[2667] := 16#5714;
   // GBK_TO_UNICODE[2668] := 16#8843;
   // GBK_TO_UNICODE[2669] := 16#5715;
   // GBK_TO_UNICODE[2670] := 16#8844;
   // GBK_TO_UNICODE[2671] := 16#5716;
   // GBK_TO_UNICODE[2672] := 16#8845;
   // GBK_TO_UNICODE[2673] := 16#5717;
   // GBK_TO_UNICODE[2674] := 16#8846;
   // GBK_TO_UNICODE[2675] := 16#5718;
   // GBK_TO_UNICODE[2676] := 16#8847;
   // GBK_TO_UNICODE[2677] := 16#5719;
   // GBK_TO_UNICODE[2678] := 16#8848;
   // GBK_TO_UNICODE[2679] := 16#571A;
   // GBK_TO_UNICODE[2680] := 16#8849;
   // GBK_TO_UNICODE[2681] := 16#571B;
   // GBK_TO_UNICODE[2682] := 16#884A;
   // GBK_TO_UNICODE[2683] := 16#571D;
   // GBK_TO_UNICODE[2684] := 16#884B;
   // GBK_TO_UNICODE[2685] := 16#571E;
   // GBK_TO_UNICODE[2686] := 16#884C;
   // GBK_TO_UNICODE[2687] := 16#5720;
   // GBK_TO_UNICODE[2688] := 16#884D;
   // GBK_TO_UNICODE[2689] := 16#5721;
   // GBK_TO_UNICODE[2690] := 16#884E;
   // GBK_TO_UNICODE[2691] := 16#5722;
   // GBK_TO_UNICODE[2692] := 16#884F;
   // GBK_TO_UNICODE[2693] := 16#5724;
   // GBK_TO_UNICODE[2694] := 16#8850;
   // GBK_TO_UNICODE[2695] := 16#5725;
   // GBK_TO_UNICODE[2696] := 16#8851;
   // GBK_TO_UNICODE[2697] := 16#5726;
   // GBK_TO_UNICODE[2698] := 16#8852;
   // GBK_TO_UNICODE[2699] := 16#5727;
   // GBK_TO_UNICODE[2700] := 16#8853;
   // GBK_TO_UNICODE[2701] := 16#572B;
   // GBK_TO_UNICODE[2702] := 16#8854;
   // GBK_TO_UNICODE[2703] := 16#5731;
   // GBK_TO_UNICODE[2704] := 16#8855;
   // GBK_TO_UNICODE[2705] := 16#5732;
   // GBK_TO_UNICODE[2706] := 16#8856;
   // GBK_TO_UNICODE[2707] := 16#5734;
   // GBK_TO_UNICODE[2708] := 16#8857;
   // GBK_TO_UNICODE[2709] := 16#5735;
   // GBK_TO_UNICODE[2710] := 16#8858;
   // GBK_TO_UNICODE[2711] := 16#5736;
   // GBK_TO_UNICODE[2712] := 16#8859;
   // GBK_TO_UNICODE[2713] := 16#5737;
   // GBK_TO_UNICODE[2714] := 16#885A;
   // GBK_TO_UNICODE[2715] := 16#5738;
   // GBK_TO_UNICODE[2716] := 16#885B;
   // GBK_TO_UNICODE[2717] := 16#573C;
   // GBK_TO_UNICODE[2718] := 16#885C;
   // GBK_TO_UNICODE[2719] := 16#573D;
   // GBK_TO_UNICODE[2720] := 16#885D;
   // GBK_TO_UNICODE[2721] := 16#573F;
   // GBK_TO_UNICODE[2722] := 16#885E;
   // GBK_TO_UNICODE[2723] := 16#5741;
   // GBK_TO_UNICODE[2724] := 16#885F;
   // GBK_TO_UNICODE[2725] := 16#5743;
   // GBK_TO_UNICODE[2726] := 16#8860;
   // GBK_TO_UNICODE[2727] := 16#5744;
   // GBK_TO_UNICODE[2728] := 16#8861;
   // GBK_TO_UNICODE[2729] := 16#5745;
   // GBK_TO_UNICODE[2730] := 16#8862;
   // GBK_TO_UNICODE[2731] := 16#5746;
   // GBK_TO_UNICODE[2732] := 16#8863;
   // GBK_TO_UNICODE[2733] := 16#5748;
   // GBK_TO_UNICODE[2734] := 16#8864;
   // GBK_TO_UNICODE[2735] := 16#5749;
   // GBK_TO_UNICODE[2736] := 16#8865;
   // GBK_TO_UNICODE[2737] := 16#574B;
   // GBK_TO_UNICODE[2738] := 16#8866;
   // GBK_TO_UNICODE[2739] := 16#5752;
   // GBK_TO_UNICODE[2740] := 16#8867;
   // GBK_TO_UNICODE[2741] := 16#5753;
   // GBK_TO_UNICODE[2742] := 16#8868;
   // GBK_TO_UNICODE[2743] := 16#5754;
   // GBK_TO_UNICODE[2744] := 16#8869;
   // GBK_TO_UNICODE[2745] := 16#5755;
   // GBK_TO_UNICODE[2746] := 16#886A;
   // GBK_TO_UNICODE[2747] := 16#5756;
   // GBK_TO_UNICODE[2748] := 16#886B;
   // GBK_TO_UNICODE[2749] := 16#5758;
   // GBK_TO_UNICODE[2750] := 16#886C;
   // GBK_TO_UNICODE[2751] := 16#5759;
   // GBK_TO_UNICODE[2752] := 16#886D;
   // GBK_TO_UNICODE[2753] := 16#5762;
   // GBK_TO_UNICODE[2754] := 16#886E;
   // GBK_TO_UNICODE[2755] := 16#5763;
   // GBK_TO_UNICODE[2756] := 16#886F;
   // GBK_TO_UNICODE[2757] := 16#5765;
   // GBK_TO_UNICODE[2758] := 16#8870;
   // GBK_TO_UNICODE[2759] := 16#5767;
   // GBK_TO_UNICODE[2760] := 16#8871;
   // GBK_TO_UNICODE[2761] := 16#576C;
   // GBK_TO_UNICODE[2762] := 16#8872;
   // GBK_TO_UNICODE[2763] := 16#576E;
   // GBK_TO_UNICODE[2764] := 16#8873;
   // GBK_TO_UNICODE[2765] := 16#5770;
   // GBK_TO_UNICODE[2766] := 16#8874;
   // GBK_TO_UNICODE[2767] := 16#5771;
   // GBK_TO_UNICODE[2768] := 16#8875;
   // GBK_TO_UNICODE[2769] := 16#5772;
   // GBK_TO_UNICODE[2770] := 16#8876;
   // GBK_TO_UNICODE[2771] := 16#5774;
   // GBK_TO_UNICODE[2772] := 16#8877;
   // GBK_TO_UNICODE[2773] := 16#5775;
   // GBK_TO_UNICODE[2774] := 16#8878;
   // GBK_TO_UNICODE[2775] := 16#5778;
   // GBK_TO_UNICODE[2776] := 16#8879;
   // GBK_TO_UNICODE[2777] := 16#5779;
   // GBK_TO_UNICODE[2778] := 16#887A;
   // GBK_TO_UNICODE[2779] := 16#577A;
   // GBK_TO_UNICODE[2780] := 16#887B;
   // GBK_TO_UNICODE[2781] := 16#577D;
   // GBK_TO_UNICODE[2782] := 16#887C;
   // GBK_TO_UNICODE[2783] := 16#577E;
   // GBK_TO_UNICODE[2784] := 16#887D;
   // GBK_TO_UNICODE[2785] := 16#577F;
   // GBK_TO_UNICODE[2786] := 16#887E;
   // GBK_TO_UNICODE[2787] := 16#5780;
   // GBK_TO_UNICODE[2788] := 16#8880;
   // GBK_TO_UNICODE[2789] := 16#5781;
   // GBK_TO_UNICODE[2790] := 16#8881;
   // GBK_TO_UNICODE[2791] := 16#5787;
   // GBK_TO_UNICODE[2792] := 16#8882;
   // GBK_TO_UNICODE[2793] := 16#5788;
   // GBK_TO_UNICODE[2794] := 16#8883;
   // GBK_TO_UNICODE[2795] := 16#5789;
   // GBK_TO_UNICODE[2796] := 16#8884;
   // GBK_TO_UNICODE[2797] := 16#578A;
   // GBK_TO_UNICODE[2798] := 16#8885;
   // GBK_TO_UNICODE[2799] := 16#578D;
   // GBK_TO_UNICODE[2800] := 16#8886;
   // GBK_TO_UNICODE[2801] := 16#578E;
   // GBK_TO_UNICODE[2802] := 16#8887;
   // GBK_TO_UNICODE[2803] := 16#578F;
   // GBK_TO_UNICODE[2804] := 16#8888;
   // GBK_TO_UNICODE[2805] := 16#5790;
   // GBK_TO_UNICODE[2806] := 16#8889;
   // GBK_TO_UNICODE[2807] := 16#5791;
   // GBK_TO_UNICODE[2808] := 16#888A;
   // GBK_TO_UNICODE[2809] := 16#5794;
   // GBK_TO_UNICODE[2810] := 16#888B;
   // GBK_TO_UNICODE[2811] := 16#5795;
   // GBK_TO_UNICODE[2812] := 16#888C;
   // GBK_TO_UNICODE[2813] := 16#5796;
   // GBK_TO_UNICODE[2814] := 16#888D;
   // GBK_TO_UNICODE[2815] := 16#5797;
   // GBK_TO_UNICODE[2816] := 16#888E;
   // GBK_TO_UNICODE[2817] := 16#5798;
   // GBK_TO_UNICODE[2818] := 16#888F;
   // GBK_TO_UNICODE[2819] := 16#5799;
   // GBK_TO_UNICODE[2820] := 16#8890;
   // GBK_TO_UNICODE[2821] := 16#579A;
   // GBK_TO_UNICODE[2822] := 16#8891;
   // GBK_TO_UNICODE[2823] := 16#579C;
   // GBK_TO_UNICODE[2824] := 16#8892;
   // GBK_TO_UNICODE[2825] := 16#579D;
   // GBK_TO_UNICODE[2826] := 16#8893;
   // GBK_TO_UNICODE[2827] := 16#579E;
   // GBK_TO_UNICODE[2828] := 16#8894;
   // GBK_TO_UNICODE[2829] := 16#579F;
   // GBK_TO_UNICODE[2830] := 16#8895;
   // GBK_TO_UNICODE[2831] := 16#57A5;
   // GBK_TO_UNICODE[2832] := 16#8896;
   // GBK_TO_UNICODE[2833] := 16#57A8;
   // GBK_TO_UNICODE[2834] := 16#8897;
   // GBK_TO_UNICODE[2835] := 16#57AA;
   // GBK_TO_UNICODE[2836] := 16#8898;
   // GBK_TO_UNICODE[2837] := 16#57AC;
   // GBK_TO_UNICODE[2838] := 16#8899;
   // GBK_TO_UNICODE[2839] := 16#57AF;
   // GBK_TO_UNICODE[2840] := 16#889A;
   // GBK_TO_UNICODE[2841] := 16#57B0;
   // GBK_TO_UNICODE[2842] := 16#889B;
   // GBK_TO_UNICODE[2843] := 16#57B1;
   // GBK_TO_UNICODE[2844] := 16#889C;
   // GBK_TO_UNICODE[2845] := 16#57B3;
   // GBK_TO_UNICODE[2846] := 16#889D;
   // GBK_TO_UNICODE[2847] := 16#57B5;
   // GBK_TO_UNICODE[2848] := 16#889E;
   // GBK_TO_UNICODE[2849] := 16#57B6;
   // GBK_TO_UNICODE[2850] := 16#889F;
   // GBK_TO_UNICODE[2851] := 16#57B7;
   // GBK_TO_UNICODE[2852] := 16#88A0;
   // GBK_TO_UNICODE[2853] := 16#57B9;
   // GBK_TO_UNICODE[2854] := 16#88A1;
   // GBK_TO_UNICODE[2855] := 16#57BA;
   // GBK_TO_UNICODE[2856] := 16#88A2;
   // GBK_TO_UNICODE[2857] := 16#57BB;
   // GBK_TO_UNICODE[2858] := 16#88A3;
   // GBK_TO_UNICODE[2859] := 16#57BC;
   // GBK_TO_UNICODE[2860] := 16#88A4;
   // GBK_TO_UNICODE[2861] := 16#57BD;
   // GBK_TO_UNICODE[2862] := 16#88A5;
   // GBK_TO_UNICODE[2863] := 16#57BE;
   // GBK_TO_UNICODE[2864] := 16#88A6;
   // GBK_TO_UNICODE[2865] := 16#57BF;
   // GBK_TO_UNICODE[2866] := 16#88A7;
   // GBK_TO_UNICODE[2867] := 16#57C0;
   // GBK_TO_UNICODE[2868] := 16#88A8;
   // GBK_TO_UNICODE[2869] := 16#57C1;
   // GBK_TO_UNICODE[2870] := 16#88A9;
   // GBK_TO_UNICODE[2871] := 16#57C4;
   // GBK_TO_UNICODE[2872] := 16#88AA;
   // GBK_TO_UNICODE[2873] := 16#57C5;
   // GBK_TO_UNICODE[2874] := 16#88AB;
   // GBK_TO_UNICODE[2875] := 16#57C6;
   // GBK_TO_UNICODE[2876] := 16#88AC;
   // GBK_TO_UNICODE[2877] := 16#57C7;
   // GBK_TO_UNICODE[2878] := 16#88AD;
   // GBK_TO_UNICODE[2879] := 16#57C8;
   // GBK_TO_UNICODE[2880] := 16#88AE;
   // GBK_TO_UNICODE[2881] := 16#57C9;
   // GBK_TO_UNICODE[2882] := 16#88AF;
   // GBK_TO_UNICODE[2883] := 16#57CA;
   // GBK_TO_UNICODE[2884] := 16#88B0;
   // GBK_TO_UNICODE[2885] := 16#57CC;
   // GBK_TO_UNICODE[2886] := 16#88B1;
   // GBK_TO_UNICODE[2887] := 16#57CD;
   // GBK_TO_UNICODE[2888] := 16#88B2;
   // GBK_TO_UNICODE[2889] := 16#57D0;
   // GBK_TO_UNICODE[2890] := 16#88B3;
   // GBK_TO_UNICODE[2891] := 16#57D1;
   // GBK_TO_UNICODE[2892] := 16#88B4;
   // GBK_TO_UNICODE[2893] := 16#57D3;
   // GBK_TO_UNICODE[2894] := 16#88B5;
   // GBK_TO_UNICODE[2895] := 16#57D6;
   // GBK_TO_UNICODE[2896] := 16#88B6;
   // GBK_TO_UNICODE[2897] := 16#57D7;
   // GBK_TO_UNICODE[2898] := 16#88B7;
   // GBK_TO_UNICODE[2899] := 16#57DB;
   // GBK_TO_UNICODE[2900] := 16#88B8;
   // GBK_TO_UNICODE[2901] := 16#57DC;
   // GBK_TO_UNICODE[2902] := 16#88B9;
   // GBK_TO_UNICODE[2903] := 16#57DE;
   // GBK_TO_UNICODE[2904] := 16#88BA;
   // GBK_TO_UNICODE[2905] := 16#57E1;
   // GBK_TO_UNICODE[2906] := 16#88BB;
   // GBK_TO_UNICODE[2907] := 16#57E2;
   // GBK_TO_UNICODE[2908] := 16#88BC;
   // GBK_TO_UNICODE[2909] := 16#57E3;
   // GBK_TO_UNICODE[2910] := 16#88BD;
   // GBK_TO_UNICODE[2911] := 16#57E5;
   // GBK_TO_UNICODE[2912] := 16#88BE;
   // GBK_TO_UNICODE[2913] := 16#57E6;
   // GBK_TO_UNICODE[2914] := 16#88BF;
   // GBK_TO_UNICODE[2915] := 16#57E7;
   // GBK_TO_UNICODE[2916] := 16#88C0;
   // GBK_TO_UNICODE[2917] := 16#57E8;
   // GBK_TO_UNICODE[2918] := 16#88C1;
   // GBK_TO_UNICODE[2919] := 16#57E9;
   // GBK_TO_UNICODE[2920] := 16#88C2;
   // GBK_TO_UNICODE[2921] := 16#57EA;
   // GBK_TO_UNICODE[2922] := 16#88C3;
   // GBK_TO_UNICODE[2923] := 16#57EB;
   // GBK_TO_UNICODE[2924] := 16#88C4;
   // GBK_TO_UNICODE[2925] := 16#57EC;
   // GBK_TO_UNICODE[2926] := 16#88C5;
   // GBK_TO_UNICODE[2927] := 16#57EE;
   // GBK_TO_UNICODE[2928] := 16#88C6;
   // GBK_TO_UNICODE[2929] := 16#57F0;
   // GBK_TO_UNICODE[2930] := 16#88C7;
   // GBK_TO_UNICODE[2931] := 16#57F1;
   // GBK_TO_UNICODE[2932] := 16#88C8;
   // GBK_TO_UNICODE[2933] := 16#57F2;
   // GBK_TO_UNICODE[2934] := 16#88C9;
   // GBK_TO_UNICODE[2935] := 16#57F3;
   // GBK_TO_UNICODE[2936] := 16#88CA;
   // GBK_TO_UNICODE[2937] := 16#57F5;
   // GBK_TO_UNICODE[2938] := 16#88CB;
   // GBK_TO_UNICODE[2939] := 16#57F6;
   // GBK_TO_UNICODE[2940] := 16#88CC;
   // GBK_TO_UNICODE[2941] := 16#57F7;
   // GBK_TO_UNICODE[2942] := 16#88CD;
   // GBK_TO_UNICODE[2943] := 16#57FB;
   // GBK_TO_UNICODE[2944] := 16#88CE;
   // GBK_TO_UNICODE[2945] := 16#57FC;
   // GBK_TO_UNICODE[2946] := 16#88CF;
   // GBK_TO_UNICODE[2947] := 16#57FE;
   // GBK_TO_UNICODE[2948] := 16#88D0;
   // GBK_TO_UNICODE[2949] := 16#57FF;
   // GBK_TO_UNICODE[2950] := 16#88D1;
   // GBK_TO_UNICODE[2951] := 16#5801;
   // GBK_TO_UNICODE[2952] := 16#88D2;
   // GBK_TO_UNICODE[2953] := 16#5803;
   // GBK_TO_UNICODE[2954] := 16#88D3;
   // GBK_TO_UNICODE[2955] := 16#5804;
   // GBK_TO_UNICODE[2956] := 16#88D4;
   // GBK_TO_UNICODE[2957] := 16#5805;
   // GBK_TO_UNICODE[2958] := 16#88D5;
   // GBK_TO_UNICODE[2959] := 16#5808;
   // GBK_TO_UNICODE[2960] := 16#88D6;
   // GBK_TO_UNICODE[2961] := 16#5809;
   // GBK_TO_UNICODE[2962] := 16#88D7;
   // GBK_TO_UNICODE[2963] := 16#580A;
   // GBK_TO_UNICODE[2964] := 16#88D8;
   // GBK_TO_UNICODE[2965] := 16#580C;
   // GBK_TO_UNICODE[2966] := 16#88D9;
   // GBK_TO_UNICODE[2967] := 16#580E;
   // GBK_TO_UNICODE[2968] := 16#88DA;
   // GBK_TO_UNICODE[2969] := 16#580F;
   // GBK_TO_UNICODE[2970] := 16#88DB;
   // GBK_TO_UNICODE[2971] := 16#5810;
   // GBK_TO_UNICODE[2972] := 16#88DC;
   // GBK_TO_UNICODE[2973] := 16#5812;
   // GBK_TO_UNICODE[2974] := 16#88DD;
   // GBK_TO_UNICODE[2975] := 16#5813;
   // GBK_TO_UNICODE[2976] := 16#88DE;
   // GBK_TO_UNICODE[2977] := 16#5814;
   // GBK_TO_UNICODE[2978] := 16#88DF;
   // GBK_TO_UNICODE[2979] := 16#5816;
   // GBK_TO_UNICODE[2980] := 16#88E0;
   // GBK_TO_UNICODE[2981] := 16#5817;
   // GBK_TO_UNICODE[2982] := 16#88E1;
   // GBK_TO_UNICODE[2983] := 16#5818;
   // GBK_TO_UNICODE[2984] := 16#88E2;
   // GBK_TO_UNICODE[2985] := 16#581A;
   // GBK_TO_UNICODE[2986] := 16#88E3;
   // GBK_TO_UNICODE[2987] := 16#581B;
   // GBK_TO_UNICODE[2988] := 16#88E4;
   // GBK_TO_UNICODE[2989] := 16#581C;
   // GBK_TO_UNICODE[2990] := 16#88E5;
   // GBK_TO_UNICODE[2991] := 16#581D;
   // GBK_TO_UNICODE[2992] := 16#88E6;
   // GBK_TO_UNICODE[2993] := 16#581F;
   // GBK_TO_UNICODE[2994] := 16#88E7;
   // GBK_TO_UNICODE[2995] := 16#5822;
   // GBK_TO_UNICODE[2996] := 16#88E8;
   // GBK_TO_UNICODE[2997] := 16#5823;
   // GBK_TO_UNICODE[2998] := 16#88E9;
   // GBK_TO_UNICODE[2999] := 16#5825;
   // GBK_TO_UNICODE[3000] := 16#88EA;
   // GBK_TO_UNICODE[3001] := 16#5826;
   // GBK_TO_UNICODE[3002] := 16#88EB;
   // GBK_TO_UNICODE[3003] := 16#5827;
   // GBK_TO_UNICODE[3004] := 16#88EC;
   // GBK_TO_UNICODE[3005] := 16#5828;
   // GBK_TO_UNICODE[3006] := 16#88ED;
   // GBK_TO_UNICODE[3007] := 16#5829;
   // GBK_TO_UNICODE[3008] := 16#88EE;
   // GBK_TO_UNICODE[3009] := 16#582B;
   // GBK_TO_UNICODE[3010] := 16#88EF;
   // GBK_TO_UNICODE[3011] := 16#582C;
   // GBK_TO_UNICODE[3012] := 16#88F0;
   // GBK_TO_UNICODE[3013] := 16#582D;
   // GBK_TO_UNICODE[3014] := 16#88F1;
   // GBK_TO_UNICODE[3015] := 16#582E;
   // GBK_TO_UNICODE[3016] := 16#88F2;
   // GBK_TO_UNICODE[3017] := 16#582F;
   // GBK_TO_UNICODE[3018] := 16#88F3;
   // GBK_TO_UNICODE[3019] := 16#5831;
   // GBK_TO_UNICODE[3020] := 16#88F4;
   // GBK_TO_UNICODE[3021] := 16#5832;
   // GBK_TO_UNICODE[3022] := 16#88F5;
   // GBK_TO_UNICODE[3023] := 16#5833;
   // GBK_TO_UNICODE[3024] := 16#88F6;
   // GBK_TO_UNICODE[3025] := 16#5834;
   // GBK_TO_UNICODE[3026] := 16#88F7;
   // GBK_TO_UNICODE[3027] := 16#5836;
   // GBK_TO_UNICODE[3028] := 16#88F8;
   // GBK_TO_UNICODE[3029] := 16#5837;
   // GBK_TO_UNICODE[3030] := 16#88F9;
   // GBK_TO_UNICODE[3031] := 16#5838;
   // GBK_TO_UNICODE[3032] := 16#88FA;
   // GBK_TO_UNICODE[3033] := 16#5839;
   // GBK_TO_UNICODE[3034] := 16#88FB;
   // GBK_TO_UNICODE[3035] := 16#583A;
   // GBK_TO_UNICODE[3036] := 16#88FC;
   // GBK_TO_UNICODE[3037] := 16#583B;
   // GBK_TO_UNICODE[3038] := 16#88FD;
   // GBK_TO_UNICODE[3039] := 16#583C;
   // GBK_TO_UNICODE[3040] := 16#88FE;
   // GBK_TO_UNICODE[3041] := 16#583D;
   // GBK_TO_UNICODE[3042] := 16#8940;
   // GBK_TO_UNICODE[3043] := 16#583E;
   // GBK_TO_UNICODE[3044] := 16#8941;
   // GBK_TO_UNICODE[3045] := 16#583F;
   // GBK_TO_UNICODE[3046] := 16#8942;
   // GBK_TO_UNICODE[3047] := 16#5840;
   // GBK_TO_UNICODE[3048] := 16#8943;
   // GBK_TO_UNICODE[3049] := 16#5841;
   // GBK_TO_UNICODE[3050] := 16#8944;
   // GBK_TO_UNICODE[3051] := 16#5842;
   // GBK_TO_UNICODE[3052] := 16#8945;
   // GBK_TO_UNICODE[3053] := 16#5843;
   // GBK_TO_UNICODE[3054] := 16#8946;
   // GBK_TO_UNICODE[3055] := 16#5845;
   // GBK_TO_UNICODE[3056] := 16#8947;
   // GBK_TO_UNICODE[3057] := 16#5846;
   // GBK_TO_UNICODE[3058] := 16#8948;
   // GBK_TO_UNICODE[3059] := 16#5847;
   // GBK_TO_UNICODE[3060] := 16#8949;
   // GBK_TO_UNICODE[3061] := 16#5848;
   // GBK_TO_UNICODE[3062] := 16#894A;
   // GBK_TO_UNICODE[3063] := 16#5849;
   // GBK_TO_UNICODE[3064] := 16#894B;
   // GBK_TO_UNICODE[3065] := 16#584A;
   // GBK_TO_UNICODE[3066] := 16#894C;
   // GBK_TO_UNICODE[3067] := 16#584B;
   // GBK_TO_UNICODE[3068] := 16#894D;
   // GBK_TO_UNICODE[3069] := 16#584E;
   // GBK_TO_UNICODE[3070] := 16#894E;
   // GBK_TO_UNICODE[3071] := 16#584F;
   // GBK_TO_UNICODE[3072] := 16#894F;
   // GBK_TO_UNICODE[3073] := 16#5850;
   // GBK_TO_UNICODE[3074] := 16#8950;
   // GBK_TO_UNICODE[3075] := 16#5852;
   // GBK_TO_UNICODE[3076] := 16#8951;
   // GBK_TO_UNICODE[3077] := 16#5853;
   // GBK_TO_UNICODE[3078] := 16#8952;
   // GBK_TO_UNICODE[3079] := 16#5855;
   // GBK_TO_UNICODE[3080] := 16#8953;
   // GBK_TO_UNICODE[3081] := 16#5856;
   // GBK_TO_UNICODE[3082] := 16#8954;
   // GBK_TO_UNICODE[3083] := 16#5857;
   // GBK_TO_UNICODE[3084] := 16#8955;
   // GBK_TO_UNICODE[3085] := 16#5859;
   // GBK_TO_UNICODE[3086] := 16#8956;
   // GBK_TO_UNICODE[3087] := 16#585A;
   // GBK_TO_UNICODE[3088] := 16#8957;
   // GBK_TO_UNICODE[3089] := 16#585B;
   // GBK_TO_UNICODE[3090] := 16#8958;
   // GBK_TO_UNICODE[3091] := 16#585C;
   // GBK_TO_UNICODE[3092] := 16#8959;
   // GBK_TO_UNICODE[3093] := 16#585D;
   // GBK_TO_UNICODE[3094] := 16#895A;
   // GBK_TO_UNICODE[3095] := 16#585F;
   // GBK_TO_UNICODE[3096] := 16#895B;
   // GBK_TO_UNICODE[3097] := 16#5860;
   // GBK_TO_UNICODE[3098] := 16#895C;
   // GBK_TO_UNICODE[3099] := 16#5861;
   // GBK_TO_UNICODE[3100] := 16#895D;
   // GBK_TO_UNICODE[3101] := 16#5862;
   // GBK_TO_UNICODE[3102] := 16#895E;
   // GBK_TO_UNICODE[3103] := 16#5863;
   // GBK_TO_UNICODE[3104] := 16#895F;
   // GBK_TO_UNICODE[3105] := 16#5864;
   // GBK_TO_UNICODE[3106] := 16#8960;
   // GBK_TO_UNICODE[3107] := 16#5866;
   // GBK_TO_UNICODE[3108] := 16#8961;
   // GBK_TO_UNICODE[3109] := 16#5867;
   // GBK_TO_UNICODE[3110] := 16#8962;
   // GBK_TO_UNICODE[3111] := 16#5868;
   // GBK_TO_UNICODE[3112] := 16#8963;
   // GBK_TO_UNICODE[3113] := 16#5869;
   // GBK_TO_UNICODE[3114] := 16#8964;
   // GBK_TO_UNICODE[3115] := 16#586A;
   // GBK_TO_UNICODE[3116] := 16#8965;
   // GBK_TO_UNICODE[3117] := 16#586D;
   // GBK_TO_UNICODE[3118] := 16#8966;
   // GBK_TO_UNICODE[3119] := 16#586E;
   // GBK_TO_UNICODE[3120] := 16#8967;
   // GBK_TO_UNICODE[3121] := 16#586F;
   // GBK_TO_UNICODE[3122] := 16#8968;
   // GBK_TO_UNICODE[3123] := 16#5870;
   // GBK_TO_UNICODE[3124] := 16#8969;
   // GBK_TO_UNICODE[3125] := 16#5871;
   // GBK_TO_UNICODE[3126] := 16#896A;
   // GBK_TO_UNICODE[3127] := 16#5872;
   // GBK_TO_UNICODE[3128] := 16#896B;
   // GBK_TO_UNICODE[3129] := 16#5873;
   // GBK_TO_UNICODE[3130] := 16#896C;
   // GBK_TO_UNICODE[3131] := 16#5874;
   // GBK_TO_UNICODE[3132] := 16#896D;
   // GBK_TO_UNICODE[3133] := 16#5875;
   // GBK_TO_UNICODE[3134] := 16#896E;
   // GBK_TO_UNICODE[3135] := 16#5876;
   // GBK_TO_UNICODE[3136] := 16#896F;
   // GBK_TO_UNICODE[3137] := 16#5877;
   // GBK_TO_UNICODE[3138] := 16#8970;
   // GBK_TO_UNICODE[3139] := 16#5878;
   // GBK_TO_UNICODE[3140] := 16#8971;
   // GBK_TO_UNICODE[3141] := 16#5879;
   // GBK_TO_UNICODE[3142] := 16#8972;
   // GBK_TO_UNICODE[3143] := 16#587A;
   // GBK_TO_UNICODE[3144] := 16#8973;
   // GBK_TO_UNICODE[3145] := 16#587B;
   // GBK_TO_UNICODE[3146] := 16#8974;
   // GBK_TO_UNICODE[3147] := 16#587C;
   // GBK_TO_UNICODE[3148] := 16#8975;
   // GBK_TO_UNICODE[3149] := 16#587D;
   // GBK_TO_UNICODE[3150] := 16#8976;
   // GBK_TO_UNICODE[3151] := 16#587F;
   // GBK_TO_UNICODE[3152] := 16#8977;
   // GBK_TO_UNICODE[3153] := 16#5882;
   // GBK_TO_UNICODE[3154] := 16#8978;
   // GBK_TO_UNICODE[3155] := 16#5884;
   // GBK_TO_UNICODE[3156] := 16#8979;
   // GBK_TO_UNICODE[3157] := 16#5886;
   // GBK_TO_UNICODE[3158] := 16#897A;
   // GBK_TO_UNICODE[3159] := 16#5887;
   // GBK_TO_UNICODE[3160] := 16#897B;
   // GBK_TO_UNICODE[3161] := 16#5888;
   // GBK_TO_UNICODE[3162] := 16#897C;
   // GBK_TO_UNICODE[3163] := 16#588A;
   // GBK_TO_UNICODE[3164] := 16#897D;
   // GBK_TO_UNICODE[3165] := 16#588B;
   // GBK_TO_UNICODE[3166] := 16#897E;
   // GBK_TO_UNICODE[3167] := 16#588C;
   // GBK_TO_UNICODE[3168] := 16#8980;
   // GBK_TO_UNICODE[3169] := 16#588D;
   // GBK_TO_UNICODE[3170] := 16#8981;
   // GBK_TO_UNICODE[3171] := 16#588E;
   // GBK_TO_UNICODE[3172] := 16#8982;
   // GBK_TO_UNICODE[3173] := 16#588F;
   // GBK_TO_UNICODE[3174] := 16#8983;
   // GBK_TO_UNICODE[3175] := 16#5890;
   // GBK_TO_UNICODE[3176] := 16#8984;
   // GBK_TO_UNICODE[3177] := 16#5891;
   // GBK_TO_UNICODE[3178] := 16#8985;
   // GBK_TO_UNICODE[3179] := 16#5894;
   // GBK_TO_UNICODE[3180] := 16#8986;
   // GBK_TO_UNICODE[3181] := 16#5895;
   // GBK_TO_UNICODE[3182] := 16#8987;
   // GBK_TO_UNICODE[3183] := 16#5896;
   // GBK_TO_UNICODE[3184] := 16#8988;
   // GBK_TO_UNICODE[3185] := 16#5897;
   // GBK_TO_UNICODE[3186] := 16#8989;
   // GBK_TO_UNICODE[3187] := 16#5898;
   // GBK_TO_UNICODE[3188] := 16#898A;
   // GBK_TO_UNICODE[3189] := 16#589B;
   // GBK_TO_UNICODE[3190] := 16#898B;
   // GBK_TO_UNICODE[3191] := 16#589C;
   // GBK_TO_UNICODE[3192] := 16#898C;
   // GBK_TO_UNICODE[3193] := 16#589D;
   // GBK_TO_UNICODE[3194] := 16#898D;
   // GBK_TO_UNICODE[3195] := 16#58A0;
   // GBK_TO_UNICODE[3196] := 16#898E;
   // GBK_TO_UNICODE[3197] := 16#58A1;
   // GBK_TO_UNICODE[3198] := 16#898F;
   // GBK_TO_UNICODE[3199] := 16#58A2;
   // GBK_TO_UNICODE[3200] := 16#8990;
   // GBK_TO_UNICODE[3201] := 16#58A3;
   // GBK_TO_UNICODE[3202] := 16#8991;
   // GBK_TO_UNICODE[3203] := 16#58A4;
   // GBK_TO_UNICODE[3204] := 16#8992;
   // GBK_TO_UNICODE[3205] := 16#58A5;
   // GBK_TO_UNICODE[3206] := 16#8993;
   // GBK_TO_UNICODE[3207] := 16#58A6;
   // GBK_TO_UNICODE[3208] := 16#8994;
   // GBK_TO_UNICODE[3209] := 16#58A7;
   // GBK_TO_UNICODE[3210] := 16#8995;
   // GBK_TO_UNICODE[3211] := 16#58AA;
   // GBK_TO_UNICODE[3212] := 16#8996;
   // GBK_TO_UNICODE[3213] := 16#58AB;
   // GBK_TO_UNICODE[3214] := 16#8997;
   // GBK_TO_UNICODE[3215] := 16#58AC;
   // GBK_TO_UNICODE[3216] := 16#8998;
   // GBK_TO_UNICODE[3217] := 16#58AD;
   // GBK_TO_UNICODE[3218] := 16#8999;
   // GBK_TO_UNICODE[3219] := 16#58AE;
   // GBK_TO_UNICODE[3220] := 16#899A;
   // GBK_TO_UNICODE[3221] := 16#58AF;
   // GBK_TO_UNICODE[3222] := 16#899B;
   // GBK_TO_UNICODE[3223] := 16#58B0;
   // GBK_TO_UNICODE[3224] := 16#899C;
   // GBK_TO_UNICODE[3225] := 16#58B1;
   // GBK_TO_UNICODE[3226] := 16#899D;
   // GBK_TO_UNICODE[3227] := 16#58B2;
   // GBK_TO_UNICODE[3228] := 16#899E;
   // GBK_TO_UNICODE[3229] := 16#58B3;
   // GBK_TO_UNICODE[3230] := 16#899F;
   // GBK_TO_UNICODE[3231] := 16#58B4;
   // GBK_TO_UNICODE[3232] := 16#89A0;
   // GBK_TO_UNICODE[3233] := 16#58B5;
   // GBK_TO_UNICODE[3234] := 16#89A1;
   // GBK_TO_UNICODE[3235] := 16#58B6;
   // GBK_TO_UNICODE[3236] := 16#89A2;
   // GBK_TO_UNICODE[3237] := 16#58B7;
   // GBK_TO_UNICODE[3238] := 16#89A3;
   // GBK_TO_UNICODE[3239] := 16#58B8;
   // GBK_TO_UNICODE[3240] := 16#89A4;
   // GBK_TO_UNICODE[3241] := 16#58B9;
   // GBK_TO_UNICODE[3242] := 16#89A5;
   // GBK_TO_UNICODE[3243] := 16#58BA;
   // GBK_TO_UNICODE[3244] := 16#89A6;
   // GBK_TO_UNICODE[3245] := 16#58BB;
   // GBK_TO_UNICODE[3246] := 16#89A7;
   // GBK_TO_UNICODE[3247] := 16#58BD;
   // GBK_TO_UNICODE[3248] := 16#89A8;
   // GBK_TO_UNICODE[3249] := 16#58BE;
   // GBK_TO_UNICODE[3250] := 16#89A9;
   // GBK_TO_UNICODE[3251] := 16#58BF;
   // GBK_TO_UNICODE[3252] := 16#89AA;
   // GBK_TO_UNICODE[3253] := 16#58C0;
   // GBK_TO_UNICODE[3254] := 16#89AB;
   // GBK_TO_UNICODE[3255] := 16#58C2;
   // GBK_TO_UNICODE[3256] := 16#89AC;
   // GBK_TO_UNICODE[3257] := 16#58C3;
   // GBK_TO_UNICODE[3258] := 16#89AD;
   // GBK_TO_UNICODE[3259] := 16#58C4;
   // GBK_TO_UNICODE[3260] := 16#89AE;
   // GBK_TO_UNICODE[3261] := 16#58C6;
   // GBK_TO_UNICODE[3262] := 16#89AF;
   // GBK_TO_UNICODE[3263] := 16#58C7;
   // GBK_TO_UNICODE[3264] := 16#89B0;
   // GBK_TO_UNICODE[3265] := 16#58C8;
   // GBK_TO_UNICODE[3266] := 16#89B1;
   // GBK_TO_UNICODE[3267] := 16#58C9;
   // GBK_TO_UNICODE[3268] := 16#89B2;
   // GBK_TO_UNICODE[3269] := 16#58CA;
   // GBK_TO_UNICODE[3270] := 16#89B3;
   // GBK_TO_UNICODE[3271] := 16#58CB;
   // GBK_TO_UNICODE[3272] := 16#89B4;
   // GBK_TO_UNICODE[3273] := 16#58CC;
   // GBK_TO_UNICODE[3274] := 16#89B5;
   // GBK_TO_UNICODE[3275] := 16#58CD;
   // GBK_TO_UNICODE[3276] := 16#89B6;
   // GBK_TO_UNICODE[3277] := 16#58CE;
   // GBK_TO_UNICODE[3278] := 16#89B7;
   // GBK_TO_UNICODE[3279] := 16#58CF;
   // GBK_TO_UNICODE[3280] := 16#89B8;
   // GBK_TO_UNICODE[3281] := 16#58D0;
   // GBK_TO_UNICODE[3282] := 16#89B9;
   // GBK_TO_UNICODE[3283] := 16#58D2;
   // GBK_TO_UNICODE[3284] := 16#89BA;
   // GBK_TO_UNICODE[3285] := 16#58D3;
   // GBK_TO_UNICODE[3286] := 16#89BB;
   // GBK_TO_UNICODE[3287] := 16#58D4;
   // GBK_TO_UNICODE[3288] := 16#89BC;
   // GBK_TO_UNICODE[3289] := 16#58D6;
   // GBK_TO_UNICODE[3290] := 16#89BD;
   // GBK_TO_UNICODE[3291] := 16#58D7;
   // GBK_TO_UNICODE[3292] := 16#89BE;
   // GBK_TO_UNICODE[3293] := 16#58D8;
   // GBK_TO_UNICODE[3294] := 16#89BF;
   // GBK_TO_UNICODE[3295] := 16#58D9;
   // GBK_TO_UNICODE[3296] := 16#89C0;
   // GBK_TO_UNICODE[3297] := 16#58DA;
   // GBK_TO_UNICODE[3298] := 16#89C1;
   // GBK_TO_UNICODE[3299] := 16#58DB;
   // GBK_TO_UNICODE[3300] := 16#89C2;
   // GBK_TO_UNICODE[3301] := 16#58DC;
   // GBK_TO_UNICODE[3302] := 16#89C3;
   // GBK_TO_UNICODE[3303] := 16#58DD;
   // GBK_TO_UNICODE[3304] := 16#89C4;
   // GBK_TO_UNICODE[3305] := 16#58DE;
   // GBK_TO_UNICODE[3306] := 16#89C5;
   // GBK_TO_UNICODE[3307] := 16#58DF;
   // GBK_TO_UNICODE[3308] := 16#89C6;
   // GBK_TO_UNICODE[3309] := 16#58E0;
   // GBK_TO_UNICODE[3310] := 16#89C7;
   // GBK_TO_UNICODE[3311] := 16#58E1;
   // GBK_TO_UNICODE[3312] := 16#89C8;
   // GBK_TO_UNICODE[3313] := 16#58E2;
   // GBK_TO_UNICODE[3314] := 16#89C9;
   // GBK_TO_UNICODE[3315] := 16#58E3;
   // GBK_TO_UNICODE[3316] := 16#89CA;
   // GBK_TO_UNICODE[3317] := 16#58E5;
   // GBK_TO_UNICODE[3318] := 16#89CB;
   // GBK_TO_UNICODE[3319] := 16#58E6;
   // GBK_TO_UNICODE[3320] := 16#89CC;
   // GBK_TO_UNICODE[3321] := 16#58E7;
   // GBK_TO_UNICODE[3322] := 16#89CD;
   // GBK_TO_UNICODE[3323] := 16#58E8;
   // GBK_TO_UNICODE[3324] := 16#89CE;
   // GBK_TO_UNICODE[3325] := 16#58E9;
   // GBK_TO_UNICODE[3326] := 16#89CF;
   // GBK_TO_UNICODE[3327] := 16#58EA;
   // GBK_TO_UNICODE[3328] := 16#89D0;
   // GBK_TO_UNICODE[3329] := 16#58ED;
   // GBK_TO_UNICODE[3330] := 16#89D1;
   // GBK_TO_UNICODE[3331] := 16#58EF;
   // GBK_TO_UNICODE[3332] := 16#89D2;
   // GBK_TO_UNICODE[3333] := 16#58F1;
   // GBK_TO_UNICODE[3334] := 16#89D3;
   // GBK_TO_UNICODE[3335] := 16#58F2;
   // GBK_TO_UNICODE[3336] := 16#89D4;
   // GBK_TO_UNICODE[3337] := 16#58F4;
   // GBK_TO_UNICODE[3338] := 16#89D5;
   // GBK_TO_UNICODE[3339] := 16#58F5;
   // GBK_TO_UNICODE[3340] := 16#89D6;
   // GBK_TO_UNICODE[3341] := 16#58F7;
   // GBK_TO_UNICODE[3342] := 16#89D7;
   // GBK_TO_UNICODE[3343] := 16#58F8;
   // GBK_TO_UNICODE[3344] := 16#89D8;
   // GBK_TO_UNICODE[3345] := 16#58FA;
   // GBK_TO_UNICODE[3346] := 16#89D9;
   // GBK_TO_UNICODE[3347] := 16#58FB;
   // GBK_TO_UNICODE[3348] := 16#89DA;
   // GBK_TO_UNICODE[3349] := 16#58FC;
   // GBK_TO_UNICODE[3350] := 16#89DB;
   // GBK_TO_UNICODE[3351] := 16#58FD;
   // GBK_TO_UNICODE[3352] := 16#89DC;
   // GBK_TO_UNICODE[3353] := 16#58FE;
   // GBK_TO_UNICODE[3354] := 16#89DD;
   // GBK_TO_UNICODE[3355] := 16#58FF;
   // GBK_TO_UNICODE[3356] := 16#89DE;
   // GBK_TO_UNICODE[3357] := 16#5900;
   // GBK_TO_UNICODE[3358] := 16#89DF;
   // GBK_TO_UNICODE[3359] := 16#5901;
   // GBK_TO_UNICODE[3360] := 16#89E0;
   // GBK_TO_UNICODE[3361] := 16#5903;
   // GBK_TO_UNICODE[3362] := 16#89E1;
   // GBK_TO_UNICODE[3363] := 16#5905;
   // GBK_TO_UNICODE[3364] := 16#89E2;
   // GBK_TO_UNICODE[3365] := 16#5906;
   // GBK_TO_UNICODE[3366] := 16#89E3;
   // GBK_TO_UNICODE[3367] := 16#5908;
   // GBK_TO_UNICODE[3368] := 16#89E4;
   // GBK_TO_UNICODE[3369] := 16#5909;
   // GBK_TO_UNICODE[3370] := 16#89E5;
   // GBK_TO_UNICODE[3371] := 16#590A;
   // GBK_TO_UNICODE[3372] := 16#89E6;
   // GBK_TO_UNICODE[3373] := 16#590B;
   // GBK_TO_UNICODE[3374] := 16#89E7;
   // GBK_TO_UNICODE[3375] := 16#590C;
   // GBK_TO_UNICODE[3376] := 16#89E8;
   // GBK_TO_UNICODE[3377] := 16#590E;
   // GBK_TO_UNICODE[3378] := 16#89E9;
   // GBK_TO_UNICODE[3379] := 16#5910;
   // GBK_TO_UNICODE[3380] := 16#89EA;
   // GBK_TO_UNICODE[3381] := 16#5911;
   // GBK_TO_UNICODE[3382] := 16#89EB;
   // GBK_TO_UNICODE[3383] := 16#5912;
   // GBK_TO_UNICODE[3384] := 16#89EC;
   // GBK_TO_UNICODE[3385] := 16#5913;
   // GBK_TO_UNICODE[3386] := 16#89ED;
   // GBK_TO_UNICODE[3387] := 16#5917;
   // GBK_TO_UNICODE[3388] := 16#89EE;
   // GBK_TO_UNICODE[3389] := 16#5918;
   // GBK_TO_UNICODE[3390] := 16#89EF;
   // GBK_TO_UNICODE[3391] := 16#591B;
   // GBK_TO_UNICODE[3392] := 16#89F0;
   // GBK_TO_UNICODE[3393] := 16#591D;
   // GBK_TO_UNICODE[3394] := 16#89F1;
   // GBK_TO_UNICODE[3395] := 16#591E;
   // GBK_TO_UNICODE[3396] := 16#89F2;
   // GBK_TO_UNICODE[3397] := 16#5920;
   // GBK_TO_UNICODE[3398] := 16#89F3;
   // GBK_TO_UNICODE[3399] := 16#5921;
   // GBK_TO_UNICODE[3400] := 16#89F4;
   // GBK_TO_UNICODE[3401] := 16#5922;
   // GBK_TO_UNICODE[3402] := 16#89F5;
   // GBK_TO_UNICODE[3403] := 16#5923;
   // GBK_TO_UNICODE[3404] := 16#89F6;
   // GBK_TO_UNICODE[3405] := 16#5926;
   // GBK_TO_UNICODE[3406] := 16#89F7;
   // GBK_TO_UNICODE[3407] := 16#5928;
   // GBK_TO_UNICODE[3408] := 16#89F8;
   // GBK_TO_UNICODE[3409] := 16#592C;
   // GBK_TO_UNICODE[3410] := 16#89F9;
   // GBK_TO_UNICODE[3411] := 16#5930;
   // GBK_TO_UNICODE[3412] := 16#89FA;
   // GBK_TO_UNICODE[3413] := 16#5932;
   // GBK_TO_UNICODE[3414] := 16#89FB;
   // GBK_TO_UNICODE[3415] := 16#5933;
   // GBK_TO_UNICODE[3416] := 16#89FC;
   // GBK_TO_UNICODE[3417] := 16#5935;
   // GBK_TO_UNICODE[3418] := 16#89FD;
   // GBK_TO_UNICODE[3419] := 16#5936;
   // GBK_TO_UNICODE[3420] := 16#89FE;
   // GBK_TO_UNICODE[3421] := 16#593B;
   // GBK_TO_UNICODE[3422] := 16#8A40;
   // GBK_TO_UNICODE[3423] := 16#593D;
   // GBK_TO_UNICODE[3424] := 16#8A41;
   // GBK_TO_UNICODE[3425] := 16#593E;
   // GBK_TO_UNICODE[3426] := 16#8A42;
   // GBK_TO_UNICODE[3427] := 16#593F;
   // GBK_TO_UNICODE[3428] := 16#8A43;
   // GBK_TO_UNICODE[3429] := 16#5940;
   // GBK_TO_UNICODE[3430] := 16#8A44;
   // GBK_TO_UNICODE[3431] := 16#5943;
   // GBK_TO_UNICODE[3432] := 16#8A45;
   // GBK_TO_UNICODE[3433] := 16#5945;
   // GBK_TO_UNICODE[3434] := 16#8A46;
   // GBK_TO_UNICODE[3435] := 16#5946;
   // GBK_TO_UNICODE[3436] := 16#8A47;
   // GBK_TO_UNICODE[3437] := 16#594A;
   // GBK_TO_UNICODE[3438] := 16#8A48;
   // GBK_TO_UNICODE[3439] := 16#594C;
   // GBK_TO_UNICODE[3440] := 16#8A49;
   // GBK_TO_UNICODE[3441] := 16#594D;
   // GBK_TO_UNICODE[3442] := 16#8A4A;
   // GBK_TO_UNICODE[3443] := 16#5950;
   // GBK_TO_UNICODE[3444] := 16#8A4B;
   // GBK_TO_UNICODE[3445] := 16#5952;
   // GBK_TO_UNICODE[3446] := 16#8A4C;
   // GBK_TO_UNICODE[3447] := 16#5953;
   // GBK_TO_UNICODE[3448] := 16#8A4D;
   // GBK_TO_UNICODE[3449] := 16#5959;
   // GBK_TO_UNICODE[3450] := 16#8A4E;
   // GBK_TO_UNICODE[3451] := 16#595B;
   // GBK_TO_UNICODE[3452] := 16#8A4F;
   // GBK_TO_UNICODE[3453] := 16#595C;
   // GBK_TO_UNICODE[3454] := 16#8A50;
   // GBK_TO_UNICODE[3455] := 16#595D;
   // GBK_TO_UNICODE[3456] := 16#8A51;
   // GBK_TO_UNICODE[3457] := 16#595E;
   // GBK_TO_UNICODE[3458] := 16#8A52;
   // GBK_TO_UNICODE[3459] := 16#595F;
   // GBK_TO_UNICODE[3460] := 16#8A53;
   // GBK_TO_UNICODE[3461] := 16#5961;
   // GBK_TO_UNICODE[3462] := 16#8A54;
   // GBK_TO_UNICODE[3463] := 16#5963;
   // GBK_TO_UNICODE[3464] := 16#8A55;
   // GBK_TO_UNICODE[3465] := 16#5964;
   // GBK_TO_UNICODE[3466] := 16#8A56;
   // GBK_TO_UNICODE[3467] := 16#5966;
   // GBK_TO_UNICODE[3468] := 16#8A57;
   // GBK_TO_UNICODE[3469] := 16#5967;
   // GBK_TO_UNICODE[3470] := 16#8A58;
   // GBK_TO_UNICODE[3471] := 16#5968;
   // GBK_TO_UNICODE[3472] := 16#8A59;
   // GBK_TO_UNICODE[3473] := 16#5969;
   // GBK_TO_UNICODE[3474] := 16#8A5A;
   // GBK_TO_UNICODE[3475] := 16#596A;
   // GBK_TO_UNICODE[3476] := 16#8A5B;
   // GBK_TO_UNICODE[3477] := 16#596B;
   // GBK_TO_UNICODE[3478] := 16#8A5C;
   // GBK_TO_UNICODE[3479] := 16#596C;
   // GBK_TO_UNICODE[3480] := 16#8A5D;
   // GBK_TO_UNICODE[3481] := 16#596D;
   // GBK_TO_UNICODE[3482] := 16#8A5E;
   // GBK_TO_UNICODE[3483] := 16#596E;
   // GBK_TO_UNICODE[3484] := 16#8A5F;
   // GBK_TO_UNICODE[3485] := 16#596F;
   // GBK_TO_UNICODE[3486] := 16#8A60;
   // GBK_TO_UNICODE[3487] := 16#5970;
   // GBK_TO_UNICODE[3488] := 16#8A61;
   // GBK_TO_UNICODE[3489] := 16#5971;
   // GBK_TO_UNICODE[3490] := 16#8A62;
   // GBK_TO_UNICODE[3491] := 16#5972;
   // GBK_TO_UNICODE[3492] := 16#8A63;
   // GBK_TO_UNICODE[3493] := 16#5975;
   // GBK_TO_UNICODE[3494] := 16#8A64;
   // GBK_TO_UNICODE[3495] := 16#5977;
   // GBK_TO_UNICODE[3496] := 16#8A65;
   // GBK_TO_UNICODE[3497] := 16#597A;
   // GBK_TO_UNICODE[3498] := 16#8A66;
   // GBK_TO_UNICODE[3499] := 16#597B;
   // GBK_TO_UNICODE[3500] := 16#8A67;
   // GBK_TO_UNICODE[3501] := 16#597C;
   // GBK_TO_UNICODE[3502] := 16#8A68;
   // GBK_TO_UNICODE[3503] := 16#597E;
   // GBK_TO_UNICODE[3504] := 16#8A69;
   // GBK_TO_UNICODE[3505] := 16#597F;
   // GBK_TO_UNICODE[3506] := 16#8A6A;
   // GBK_TO_UNICODE[3507] := 16#5980;
   // GBK_TO_UNICODE[3508] := 16#8A6B;
   // GBK_TO_UNICODE[3509] := 16#5985;
   // GBK_TO_UNICODE[3510] := 16#8A6C;
   // GBK_TO_UNICODE[3511] := 16#5989;
   // GBK_TO_UNICODE[3512] := 16#8A6D;
   // GBK_TO_UNICODE[3513] := 16#598B;
   // GBK_TO_UNICODE[3514] := 16#8A6E;
   // GBK_TO_UNICODE[3515] := 16#598C;
   // GBK_TO_UNICODE[3516] := 16#8A6F;
   // GBK_TO_UNICODE[3517] := 16#598E;
   // GBK_TO_UNICODE[3518] := 16#8A70;
   // GBK_TO_UNICODE[3519] := 16#598F;
   // GBK_TO_UNICODE[3520] := 16#8A71;
   // GBK_TO_UNICODE[3521] := 16#5990;
   // GBK_TO_UNICODE[3522] := 16#8A72;
   // GBK_TO_UNICODE[3523] := 16#5991;
   // GBK_TO_UNICODE[3524] := 16#8A73;
   // GBK_TO_UNICODE[3525] := 16#5994;
   // GBK_TO_UNICODE[3526] := 16#8A74;
   // GBK_TO_UNICODE[3527] := 16#5995;
   // GBK_TO_UNICODE[3528] := 16#8A75;
   // GBK_TO_UNICODE[3529] := 16#5998;
   // GBK_TO_UNICODE[3530] := 16#8A76;
   // GBK_TO_UNICODE[3531] := 16#599A;
   // GBK_TO_UNICODE[3532] := 16#8A77;
   // GBK_TO_UNICODE[3533] := 16#599B;
   // GBK_TO_UNICODE[3534] := 16#8A78;
   // GBK_TO_UNICODE[3535] := 16#599C;
   // GBK_TO_UNICODE[3536] := 16#8A79;
   // GBK_TO_UNICODE[3537] := 16#599D;
   // GBK_TO_UNICODE[3538] := 16#8A7A;
   // GBK_TO_UNICODE[3539] := 16#599F;
   // GBK_TO_UNICODE[3540] := 16#8A7B;
   // GBK_TO_UNICODE[3541] := 16#59A0;
   // GBK_TO_UNICODE[3542] := 16#8A7C;
   // GBK_TO_UNICODE[3543] := 16#59A1;
   // GBK_TO_UNICODE[3544] := 16#8A7D;
   // GBK_TO_UNICODE[3545] := 16#59A2;
   // GBK_TO_UNICODE[3546] := 16#8A7E;
   // GBK_TO_UNICODE[3547] := 16#59A6;
   // GBK_TO_UNICODE[3548] := 16#8A80;
   // GBK_TO_UNICODE[3549] := 16#59A7;
   // GBK_TO_UNICODE[3550] := 16#8A81;
   // GBK_TO_UNICODE[3551] := 16#59AC;
   // GBK_TO_UNICODE[3552] := 16#8A82;
   // GBK_TO_UNICODE[3553] := 16#59AD;
   // GBK_TO_UNICODE[3554] := 16#8A83;
   // GBK_TO_UNICODE[3555] := 16#59B0;
   // GBK_TO_UNICODE[3556] := 16#8A84;
   // GBK_TO_UNICODE[3557] := 16#59B1;
   // GBK_TO_UNICODE[3558] := 16#8A85;
   // GBK_TO_UNICODE[3559] := 16#59B3;
   // GBK_TO_UNICODE[3560] := 16#8A86;
   // GBK_TO_UNICODE[3561] := 16#59B4;
   // GBK_TO_UNICODE[3562] := 16#8A87;
   // GBK_TO_UNICODE[3563] := 16#59B5;
   // GBK_TO_UNICODE[3564] := 16#8A88;
   // GBK_TO_UNICODE[3565] := 16#59B6;
   // GBK_TO_UNICODE[3566] := 16#8A89;
   // GBK_TO_UNICODE[3567] := 16#59B7;
   // GBK_TO_UNICODE[3568] := 16#8A8A;
   // GBK_TO_UNICODE[3569] := 16#59B8;
   // GBK_TO_UNICODE[3570] := 16#8A8B;
   // GBK_TO_UNICODE[3571] := 16#59BA;
   // GBK_TO_UNICODE[3572] := 16#8A8C;
   // GBK_TO_UNICODE[3573] := 16#59BC;
   // GBK_TO_UNICODE[3574] := 16#8A8D;
   // GBK_TO_UNICODE[3575] := 16#59BD;
   // GBK_TO_UNICODE[3576] := 16#8A8E;
   // GBK_TO_UNICODE[3577] := 16#59BF;
   // GBK_TO_UNICODE[3578] := 16#8A8F;
   // GBK_TO_UNICODE[3579] := 16#59C0;
   // GBK_TO_UNICODE[3580] := 16#8A90;
   // GBK_TO_UNICODE[3581] := 16#59C1;
   // GBK_TO_UNICODE[3582] := 16#8A91;
   // GBK_TO_UNICODE[3583] := 16#59C2;
   // GBK_TO_UNICODE[3584] := 16#8A92;
   // GBK_TO_UNICODE[3585] := 16#59C3;
   // GBK_TO_UNICODE[3586] := 16#8A93;
   // GBK_TO_UNICODE[3587] := 16#59C4;
   // GBK_TO_UNICODE[3588] := 16#8A94;
   // GBK_TO_UNICODE[3589] := 16#59C5;
   // GBK_TO_UNICODE[3590] := 16#8A95;
   // GBK_TO_UNICODE[3591] := 16#59C7;
   // GBK_TO_UNICODE[3592] := 16#8A96;
   // GBK_TO_UNICODE[3593] := 16#59C8;
   // GBK_TO_UNICODE[3594] := 16#8A97;
   // GBK_TO_UNICODE[3595] := 16#59C9;
   // GBK_TO_UNICODE[3596] := 16#8A98;
   // GBK_TO_UNICODE[3597] := 16#59CC;
   // GBK_TO_UNICODE[3598] := 16#8A99;
   // GBK_TO_UNICODE[3599] := 16#59CD;
   // GBK_TO_UNICODE[3600] := 16#8A9A;
   // GBK_TO_UNICODE[3601] := 16#59CE;
   // GBK_TO_UNICODE[3602] := 16#8A9B;
   // GBK_TO_UNICODE[3603] := 16#59CF;
   // GBK_TO_UNICODE[3604] := 16#8A9C;
   // GBK_TO_UNICODE[3605] := 16#59D5;
   // GBK_TO_UNICODE[3606] := 16#8A9D;
   // GBK_TO_UNICODE[3607] := 16#59D6;
   // GBK_TO_UNICODE[3608] := 16#8A9E;
   // GBK_TO_UNICODE[3609] := 16#59D9;
   // GBK_TO_UNICODE[3610] := 16#8A9F;
   // GBK_TO_UNICODE[3611] := 16#59DB;
   // GBK_TO_UNICODE[3612] := 16#8AA0;
   // GBK_TO_UNICODE[3613] := 16#59DE;
   // GBK_TO_UNICODE[3614] := 16#8AA1;
   // GBK_TO_UNICODE[3615] := 16#59DF;
   // GBK_TO_UNICODE[3616] := 16#8AA2;
   // GBK_TO_UNICODE[3617] := 16#59E0;
   // GBK_TO_UNICODE[3618] := 16#8AA3;
   // GBK_TO_UNICODE[3619] := 16#59E1;
   // GBK_TO_UNICODE[3620] := 16#8AA4;
   // GBK_TO_UNICODE[3621] := 16#59E2;
   // GBK_TO_UNICODE[3622] := 16#8AA5;
   // GBK_TO_UNICODE[3623] := 16#59E4;
   // GBK_TO_UNICODE[3624] := 16#8AA6;
   // GBK_TO_UNICODE[3625] := 16#59E6;
   // GBK_TO_UNICODE[3626] := 16#8AA7;
   // GBK_TO_UNICODE[3627] := 16#59E7;
   // GBK_TO_UNICODE[3628] := 16#8AA8;
   // GBK_TO_UNICODE[3629] := 16#59E9;
   // GBK_TO_UNICODE[3630] := 16#8AA9;
   // GBK_TO_UNICODE[3631] := 16#59EA;
   // GBK_TO_UNICODE[3632] := 16#8AAA;
   // GBK_TO_UNICODE[3633] := 16#59EB;
   // GBK_TO_UNICODE[3634] := 16#8AAB;
   // GBK_TO_UNICODE[3635] := 16#59ED;
   // GBK_TO_UNICODE[3636] := 16#8AAC;
   // GBK_TO_UNICODE[3637] := 16#59EE;
   // GBK_TO_UNICODE[3638] := 16#8AAD;
   // GBK_TO_UNICODE[3639] := 16#59EF;
   // GBK_TO_UNICODE[3640] := 16#8AAE;
   // GBK_TO_UNICODE[3641] := 16#59F0;
   // GBK_TO_UNICODE[3642] := 16#8AAF;
   // GBK_TO_UNICODE[3643] := 16#59F1;
   // GBK_TO_UNICODE[3644] := 16#8AB0;
   // GBK_TO_UNICODE[3645] := 16#59F2;
   // GBK_TO_UNICODE[3646] := 16#8AB1;
   // GBK_TO_UNICODE[3647] := 16#59F3;
   // GBK_TO_UNICODE[3648] := 16#8AB2;
   // GBK_TO_UNICODE[3649] := 16#59F4;
   // GBK_TO_UNICODE[3650] := 16#8AB3;
   // GBK_TO_UNICODE[3651] := 16#59F5;
   // GBK_TO_UNICODE[3652] := 16#8AB4;
   // GBK_TO_UNICODE[3653] := 16#59F6;
   // GBK_TO_UNICODE[3654] := 16#8AB5;
   // GBK_TO_UNICODE[3655] := 16#59F7;
   // GBK_TO_UNICODE[3656] := 16#8AB6;
   // GBK_TO_UNICODE[3657] := 16#59F8;
   // GBK_TO_UNICODE[3658] := 16#8AB7;
   // GBK_TO_UNICODE[3659] := 16#59FA;
   // GBK_TO_UNICODE[3660] := 16#8AB8;
   // GBK_TO_UNICODE[3661] := 16#59FC;
   // GBK_TO_UNICODE[3662] := 16#8AB9;
   // GBK_TO_UNICODE[3663] := 16#59FD;
   // GBK_TO_UNICODE[3664] := 16#8ABA;
   // GBK_TO_UNICODE[3665] := 16#59FE;
   // GBK_TO_UNICODE[3666] := 16#8ABB;
   // GBK_TO_UNICODE[3667] := 16#5A00;
   // GBK_TO_UNICODE[3668] := 16#8ABC;
   // GBK_TO_UNICODE[3669] := 16#5A02;
   // GBK_TO_UNICODE[3670] := 16#8ABD;
   // GBK_TO_UNICODE[3671] := 16#5A0A;
   // GBK_TO_UNICODE[3672] := 16#8ABE;
   // GBK_TO_UNICODE[3673] := 16#5A0B;
   // GBK_TO_UNICODE[3674] := 16#8ABF;
   // GBK_TO_UNICODE[3675] := 16#5A0D;
   // GBK_TO_UNICODE[3676] := 16#8AC0;
   // GBK_TO_UNICODE[3677] := 16#5A0E;
   // GBK_TO_UNICODE[3678] := 16#8AC1;
   // GBK_TO_UNICODE[3679] := 16#5A0F;
   // GBK_TO_UNICODE[3680] := 16#8AC2;
   // GBK_TO_UNICODE[3681] := 16#5A10;
   // GBK_TO_UNICODE[3682] := 16#8AC3;
   // GBK_TO_UNICODE[3683] := 16#5A12;
   // GBK_TO_UNICODE[3684] := 16#8AC4;
   // GBK_TO_UNICODE[3685] := 16#5A14;
   // GBK_TO_UNICODE[3686] := 16#8AC5;
   // GBK_TO_UNICODE[3687] := 16#5A15;
   // GBK_TO_UNICODE[3688] := 16#8AC6;
   // GBK_TO_UNICODE[3689] := 16#5A16;
   // GBK_TO_UNICODE[3690] := 16#8AC7;
   // GBK_TO_UNICODE[3691] := 16#5A17;
   // GBK_TO_UNICODE[3692] := 16#8AC8;
   // GBK_TO_UNICODE[3693] := 16#5A19;
   // GBK_TO_UNICODE[3694] := 16#8AC9;
   // GBK_TO_UNICODE[3695] := 16#5A1A;
   // GBK_TO_UNICODE[3696] := 16#8ACA;
   // GBK_TO_UNICODE[3697] := 16#5A1B;
   // GBK_TO_UNICODE[3698] := 16#8ACB;
   // GBK_TO_UNICODE[3699] := 16#5A1D;
   // GBK_TO_UNICODE[3700] := 16#8ACC;
   // GBK_TO_UNICODE[3701] := 16#5A1E;
   // GBK_TO_UNICODE[3702] := 16#8ACD;
   // GBK_TO_UNICODE[3703] := 16#5A21;
   // GBK_TO_UNICODE[3704] := 16#8ACE;
   // GBK_TO_UNICODE[3705] := 16#5A22;
   // GBK_TO_UNICODE[3706] := 16#8ACF;
   // GBK_TO_UNICODE[3707] := 16#5A24;
   // GBK_TO_UNICODE[3708] := 16#8AD0;
   // GBK_TO_UNICODE[3709] := 16#5A26;
   // GBK_TO_UNICODE[3710] := 16#8AD1;
   // GBK_TO_UNICODE[3711] := 16#5A27;
   // GBK_TO_UNICODE[3712] := 16#8AD2;
   // GBK_TO_UNICODE[3713] := 16#5A28;
   // GBK_TO_UNICODE[3714] := 16#8AD3;
   // GBK_TO_UNICODE[3715] := 16#5A2A;
   // GBK_TO_UNICODE[3716] := 16#8AD4;
   // GBK_TO_UNICODE[3717] := 16#5A2B;
   // GBK_TO_UNICODE[3718] := 16#8AD5;
   // GBK_TO_UNICODE[3719] := 16#5A2C;
   // GBK_TO_UNICODE[3720] := 16#8AD6;
   // GBK_TO_UNICODE[3721] := 16#5A2D;
   // GBK_TO_UNICODE[3722] := 16#8AD7;
   // GBK_TO_UNICODE[3723] := 16#5A2E;
   // GBK_TO_UNICODE[3724] := 16#8AD8;
   // GBK_TO_UNICODE[3725] := 16#5A2F;
   // GBK_TO_UNICODE[3726] := 16#8AD9;
   // GBK_TO_UNICODE[3727] := 16#5A30;
   // GBK_TO_UNICODE[3728] := 16#8ADA;
   // GBK_TO_UNICODE[3729] := 16#5A33;
   // GBK_TO_UNICODE[3730] := 16#8ADB;
   // GBK_TO_UNICODE[3731] := 16#5A35;
   // GBK_TO_UNICODE[3732] := 16#8ADC;
   // GBK_TO_UNICODE[3733] := 16#5A37;
   // GBK_TO_UNICODE[3734] := 16#8ADD;
   // GBK_TO_UNICODE[3735] := 16#5A38;
   // GBK_TO_UNICODE[3736] := 16#8ADE;
   // GBK_TO_UNICODE[3737] := 16#5A39;
   // GBK_TO_UNICODE[3738] := 16#8ADF;
   // GBK_TO_UNICODE[3739] := 16#5A3A;
   // GBK_TO_UNICODE[3740] := 16#8AE0;
   // GBK_TO_UNICODE[3741] := 16#5A3B;
   // GBK_TO_UNICODE[3742] := 16#8AE1;
   // GBK_TO_UNICODE[3743] := 16#5A3D;
   // GBK_TO_UNICODE[3744] := 16#8AE2;
   // GBK_TO_UNICODE[3745] := 16#5A3E;
   // GBK_TO_UNICODE[3746] := 16#8AE3;
   // GBK_TO_UNICODE[3747] := 16#5A3F;
   // GBK_TO_UNICODE[3748] := 16#8AE4;
   // GBK_TO_UNICODE[3749] := 16#5A41;
   // GBK_TO_UNICODE[3750] := 16#8AE5;
   // GBK_TO_UNICODE[3751] := 16#5A42;
   // GBK_TO_UNICODE[3752] := 16#8AE6;
   // GBK_TO_UNICODE[3753] := 16#5A43;
   // GBK_TO_UNICODE[3754] := 16#8AE7;
   // GBK_TO_UNICODE[3755] := 16#5A44;
   // GBK_TO_UNICODE[3756] := 16#8AE8;
   // GBK_TO_UNICODE[3757] := 16#5A45;
   // GBK_TO_UNICODE[3758] := 16#8AE9;
   // GBK_TO_UNICODE[3759] := 16#5A47;
   // GBK_TO_UNICODE[3760] := 16#8AEA;
   // GBK_TO_UNICODE[3761] := 16#5A48;
   // GBK_TO_UNICODE[3762] := 16#8AEB;
   // GBK_TO_UNICODE[3763] := 16#5A4B;
   // GBK_TO_UNICODE[3764] := 16#8AEC;
   // GBK_TO_UNICODE[3765] := 16#5A4C;
   // GBK_TO_UNICODE[3766] := 16#8AED;
   // GBK_TO_UNICODE[3767] := 16#5A4D;
   // GBK_TO_UNICODE[3768] := 16#8AEE;
   // GBK_TO_UNICODE[3769] := 16#5A4E;
   // GBK_TO_UNICODE[3770] := 16#8AEF;
   // GBK_TO_UNICODE[3771] := 16#5A4F;
   // GBK_TO_UNICODE[3772] := 16#8AF0;
   // GBK_TO_UNICODE[3773] := 16#5A50;
   // GBK_TO_UNICODE[3774] := 16#8AF1;
   // GBK_TO_UNICODE[3775] := 16#5A51;
   // GBK_TO_UNICODE[3776] := 16#8AF2;
   // GBK_TO_UNICODE[3777] := 16#5A52;
   // GBK_TO_UNICODE[3778] := 16#8AF3;
   // GBK_TO_UNICODE[3779] := 16#5A53;
   // GBK_TO_UNICODE[3780] := 16#8AF4;
   // GBK_TO_UNICODE[3781] := 16#5A54;
   // GBK_TO_UNICODE[3782] := 16#8AF5;
   // GBK_TO_UNICODE[3783] := 16#5A56;
   // GBK_TO_UNICODE[3784] := 16#8AF6;
   // GBK_TO_UNICODE[3785] := 16#5A57;
   // GBK_TO_UNICODE[3786] := 16#8AF7;
   // GBK_TO_UNICODE[3787] := 16#5A58;
   // GBK_TO_UNICODE[3788] := 16#8AF8;
   // GBK_TO_UNICODE[3789] := 16#5A59;
   // GBK_TO_UNICODE[3790] := 16#8AF9;
   // GBK_TO_UNICODE[3791] := 16#5A5B;
   // GBK_TO_UNICODE[3792] := 16#8AFA;
   // GBK_TO_UNICODE[3793] := 16#5A5C;
   // GBK_TO_UNICODE[3794] := 16#8AFB;
   // GBK_TO_UNICODE[3795] := 16#5A5D;
   // GBK_TO_UNICODE[3796] := 16#8AFC;
   // GBK_TO_UNICODE[3797] := 16#5A5E;
   // GBK_TO_UNICODE[3798] := 16#8AFD;
   // GBK_TO_UNICODE[3799] := 16#5A5F;
   // GBK_TO_UNICODE[3800] := 16#8AFE;
   // GBK_TO_UNICODE[3801] := 16#5A60;
   // GBK_TO_UNICODE[3802] := 16#8B40;
   // GBK_TO_UNICODE[3803] := 16#5A61;
   // GBK_TO_UNICODE[3804] := 16#8B41;
   // GBK_TO_UNICODE[3805] := 16#5A63;
   // GBK_TO_UNICODE[3806] := 16#8B42;
   // GBK_TO_UNICODE[3807] := 16#5A64;
   // GBK_TO_UNICODE[3808] := 16#8B43;
   // GBK_TO_UNICODE[3809] := 16#5A65;
   // GBK_TO_UNICODE[3810] := 16#8B44;
   // GBK_TO_UNICODE[3811] := 16#5A66;
   // GBK_TO_UNICODE[3812] := 16#8B45;
   // GBK_TO_UNICODE[3813] := 16#5A68;
   // GBK_TO_UNICODE[3814] := 16#8B46;
   // GBK_TO_UNICODE[3815] := 16#5A69;
   // GBK_TO_UNICODE[3816] := 16#8B47;
   // GBK_TO_UNICODE[3817] := 16#5A6B;
   // GBK_TO_UNICODE[3818] := 16#8B48;
   // GBK_TO_UNICODE[3819] := 16#5A6C;
   // GBK_TO_UNICODE[3820] := 16#8B49;
   // GBK_TO_UNICODE[3821] := 16#5A6D;
   // GBK_TO_UNICODE[3822] := 16#8B4A;
   // GBK_TO_UNICODE[3823] := 16#5A6E;
   // GBK_TO_UNICODE[3824] := 16#8B4B;
   // GBK_TO_UNICODE[3825] := 16#5A6F;
   // GBK_TO_UNICODE[3826] := 16#8B4C;
   // GBK_TO_UNICODE[3827] := 16#5A70;
   // GBK_TO_UNICODE[3828] := 16#8B4D;
   // GBK_TO_UNICODE[3829] := 16#5A71;
   // GBK_TO_UNICODE[3830] := 16#8B4E;
   // GBK_TO_UNICODE[3831] := 16#5A72;
   // GBK_TO_UNICODE[3832] := 16#8B4F;
   // GBK_TO_UNICODE[3833] := 16#5A73;
   // GBK_TO_UNICODE[3834] := 16#8B50;
   // GBK_TO_UNICODE[3835] := 16#5A78;
   // GBK_TO_UNICODE[3836] := 16#8B51;
   // GBK_TO_UNICODE[3837] := 16#5A79;
   // GBK_TO_UNICODE[3838] := 16#8B52;
   // GBK_TO_UNICODE[3839] := 16#5A7B;
   // GBK_TO_UNICODE[3840] := 16#8B53;
   // GBK_TO_UNICODE[3841] := 16#5A7C;
   // GBK_TO_UNICODE[3842] := 16#8B54;
   // GBK_TO_UNICODE[3843] := 16#5A7D;
   // GBK_TO_UNICODE[3844] := 16#8B55;
   // GBK_TO_UNICODE[3845] := 16#5A7E;
   // GBK_TO_UNICODE[3846] := 16#8B56;
   // GBK_TO_UNICODE[3847] := 16#5A80;
   // GBK_TO_UNICODE[3848] := 16#8B57;
   // GBK_TO_UNICODE[3849] := 16#5A81;
   // GBK_TO_UNICODE[3850] := 16#8B58;
   // GBK_TO_UNICODE[3851] := 16#5A82;
   // GBK_TO_UNICODE[3852] := 16#8B59;
   // GBK_TO_UNICODE[3853] := 16#5A83;
   // GBK_TO_UNICODE[3854] := 16#8B5A;
   // GBK_TO_UNICODE[3855] := 16#5A84;
   // GBK_TO_UNICODE[3856] := 16#8B5B;
   // GBK_TO_UNICODE[3857] := 16#5A85;
   // GBK_TO_UNICODE[3858] := 16#8B5C;
   // GBK_TO_UNICODE[3859] := 16#5A86;
   // GBK_TO_UNICODE[3860] := 16#8B5D;
   // GBK_TO_UNICODE[3861] := 16#5A87;
   // GBK_TO_UNICODE[3862] := 16#8B5E;
   // GBK_TO_UNICODE[3863] := 16#5A88;
   // GBK_TO_UNICODE[3864] := 16#8B5F;
   // GBK_TO_UNICODE[3865] := 16#5A89;
   // GBK_TO_UNICODE[3866] := 16#8B60;
   // GBK_TO_UNICODE[3867] := 16#5A8A;
   // GBK_TO_UNICODE[3868] := 16#8B61;
   // GBK_TO_UNICODE[3869] := 16#5A8B;
   // GBK_TO_UNICODE[3870] := 16#8B62;
   // GBK_TO_UNICODE[3871] := 16#5A8C;
   // GBK_TO_UNICODE[3872] := 16#8B63;
   // GBK_TO_UNICODE[3873] := 16#5A8D;
   // GBK_TO_UNICODE[3874] := 16#8B64;
   // GBK_TO_UNICODE[3875] := 16#5A8E;
   // GBK_TO_UNICODE[3876] := 16#8B65;
   // GBK_TO_UNICODE[3877] := 16#5A8F;
   // GBK_TO_UNICODE[3878] := 16#8B66;
   // GBK_TO_UNICODE[3879] := 16#5A90;
   // GBK_TO_UNICODE[3880] := 16#8B67;
   // GBK_TO_UNICODE[3881] := 16#5A91;
   // GBK_TO_UNICODE[3882] := 16#8B68;
   // GBK_TO_UNICODE[3883] := 16#5A93;
   // GBK_TO_UNICODE[3884] := 16#8B69;
   // GBK_TO_UNICODE[3885] := 16#5A94;
   // GBK_TO_UNICODE[3886] := 16#8B6A;
   // GBK_TO_UNICODE[3887] := 16#5A95;
   // GBK_TO_UNICODE[3888] := 16#8B6B;
   // GBK_TO_UNICODE[3889] := 16#5A96;
   // GBK_TO_UNICODE[3890] := 16#8B6C;
   // GBK_TO_UNICODE[3891] := 16#5A97;
   // GBK_TO_UNICODE[3892] := 16#8B6D;
   // GBK_TO_UNICODE[3893] := 16#5A98;
   // GBK_TO_UNICODE[3894] := 16#8B6E;
   // GBK_TO_UNICODE[3895] := 16#5A99;
   // GBK_TO_UNICODE[3896] := 16#8B6F;
   // GBK_TO_UNICODE[3897] := 16#5A9C;
   // GBK_TO_UNICODE[3898] := 16#8B70;
   // GBK_TO_UNICODE[3899] := 16#5A9D;
   // GBK_TO_UNICODE[3900] := 16#8B71;
   // GBK_TO_UNICODE[3901] := 16#5A9E;
   // GBK_TO_UNICODE[3902] := 16#8B72;
   // GBK_TO_UNICODE[3903] := 16#5A9F;
   // GBK_TO_UNICODE[3904] := 16#8B73;
   // GBK_TO_UNICODE[3905] := 16#5AA0;
   // GBK_TO_UNICODE[3906] := 16#8B74;
   // GBK_TO_UNICODE[3907] := 16#5AA1;
   // GBK_TO_UNICODE[3908] := 16#8B75;
   // GBK_TO_UNICODE[3909] := 16#5AA2;
   // GBK_TO_UNICODE[3910] := 16#8B76;
   // GBK_TO_UNICODE[3911] := 16#5AA3;
   // GBK_TO_UNICODE[3912] := 16#8B77;
   // GBK_TO_UNICODE[3913] := 16#5AA4;
   // GBK_TO_UNICODE[3914] := 16#8B78;
   // GBK_TO_UNICODE[3915] := 16#5AA5;
   // GBK_TO_UNICODE[3916] := 16#8B79;
   // GBK_TO_UNICODE[3917] := 16#5AA6;
   // GBK_TO_UNICODE[3918] := 16#8B7A;
   // GBK_TO_UNICODE[3919] := 16#5AA7;
   // GBK_TO_UNICODE[3920] := 16#8B7B;
   // GBK_TO_UNICODE[3921] := 16#5AA8;
   // GBK_TO_UNICODE[3922] := 16#8B7C;
   // GBK_TO_UNICODE[3923] := 16#5AA9;
   // GBK_TO_UNICODE[3924] := 16#8B7D;
   // GBK_TO_UNICODE[3925] := 16#5AAB;
   // GBK_TO_UNICODE[3926] := 16#8B7E;
   // GBK_TO_UNICODE[3927] := 16#5AAC;
   // GBK_TO_UNICODE[3928] := 16#8B80;
   // GBK_TO_UNICODE[3929] := 16#5AAD;
   // GBK_TO_UNICODE[3930] := 16#8B81;
   // GBK_TO_UNICODE[3931] := 16#5AAE;
   // GBK_TO_UNICODE[3932] := 16#8B82;
   // GBK_TO_UNICODE[3933] := 16#5AAF;
   // GBK_TO_UNICODE[3934] := 16#8B83;
   // GBK_TO_UNICODE[3935] := 16#5AB0;
   // GBK_TO_UNICODE[3936] := 16#8B84;
   // GBK_TO_UNICODE[3937] := 16#5AB1;
   // GBK_TO_UNICODE[3938] := 16#8B85;
   // GBK_TO_UNICODE[3939] := 16#5AB4;
   // GBK_TO_UNICODE[3940] := 16#8B86;
   // GBK_TO_UNICODE[3941] := 16#5AB6;
   // GBK_TO_UNICODE[3942] := 16#8B87;
   // GBK_TO_UNICODE[3943] := 16#5AB7;
   // GBK_TO_UNICODE[3944] := 16#8B88;
   // GBK_TO_UNICODE[3945] := 16#5AB9;
   // GBK_TO_UNICODE[3946] := 16#8B89;
   // GBK_TO_UNICODE[3947] := 16#5ABA;
   // GBK_TO_UNICODE[3948] := 16#8B8A;
   // GBK_TO_UNICODE[3949] := 16#5ABB;
   // GBK_TO_UNICODE[3950] := 16#8B8B;
   // GBK_TO_UNICODE[3951] := 16#5ABC;
   // GBK_TO_UNICODE[3952] := 16#8B8C;
   // GBK_TO_UNICODE[3953] := 16#5ABD;
   // GBK_TO_UNICODE[3954] := 16#8B8D;
   // GBK_TO_UNICODE[3955] := 16#5ABF;
   // GBK_TO_UNICODE[3956] := 16#8B8E;
   // GBK_TO_UNICODE[3957] := 16#5AC0;
   // GBK_TO_UNICODE[3958] := 16#8B8F;
   // GBK_TO_UNICODE[3959] := 16#5AC3;
   // GBK_TO_UNICODE[3960] := 16#8B90;
   // GBK_TO_UNICODE[3961] := 16#5AC4;
   // GBK_TO_UNICODE[3962] := 16#8B91;
   // GBK_TO_UNICODE[3963] := 16#5AC5;
   // GBK_TO_UNICODE[3964] := 16#8B92;
   // GBK_TO_UNICODE[3965] := 16#5AC6;
   // GBK_TO_UNICODE[3966] := 16#8B93;
   // GBK_TO_UNICODE[3967] := 16#5AC7;
   // GBK_TO_UNICODE[3968] := 16#8B94;
   // GBK_TO_UNICODE[3969] := 16#5AC8;
   // GBK_TO_UNICODE[3970] := 16#8B95;
   // GBK_TO_UNICODE[3971] := 16#5ACA;
   // GBK_TO_UNICODE[3972] := 16#8B96;
   // GBK_TO_UNICODE[3973] := 16#5ACB;
   // GBK_TO_UNICODE[3974] := 16#8B97;
   // GBK_TO_UNICODE[3975] := 16#5ACD;
   // GBK_TO_UNICODE[3976] := 16#8B98;
   // GBK_TO_UNICODE[3977] := 16#5ACE;
   // GBK_TO_UNICODE[3978] := 16#8B99;
   // GBK_TO_UNICODE[3979] := 16#5ACF;
   // GBK_TO_UNICODE[3980] := 16#8B9A;
   // GBK_TO_UNICODE[3981] := 16#5AD0;
   // GBK_TO_UNICODE[3982] := 16#8B9B;
   // GBK_TO_UNICODE[3983] := 16#5AD1;
   // GBK_TO_UNICODE[3984] := 16#8B9C;
   // GBK_TO_UNICODE[3985] := 16#5AD3;
   // GBK_TO_UNICODE[3986] := 16#8B9D;
   // GBK_TO_UNICODE[3987] := 16#5AD5;
   // GBK_TO_UNICODE[3988] := 16#8B9E;
   // GBK_TO_UNICODE[3989] := 16#5AD7;
   // GBK_TO_UNICODE[3990] := 16#8B9F;
   // GBK_TO_UNICODE[3991] := 16#5AD9;
   // GBK_TO_UNICODE[3992] := 16#8BA0;
   // GBK_TO_UNICODE[3993] := 16#5ADA;
   // GBK_TO_UNICODE[3994] := 16#8BA1;
   // GBK_TO_UNICODE[3995] := 16#5ADB;
   // GBK_TO_UNICODE[3996] := 16#8BA2;
   // GBK_TO_UNICODE[3997] := 16#5ADD;
   // GBK_TO_UNICODE[3998] := 16#8BA3;
   // GBK_TO_UNICODE[3999] := 16#5ADE;
   // GBK_TO_UNICODE[4000] := 16#8BA4;
   // GBK_TO_UNICODE[4001] := 16#5ADF;
   // GBK_TO_UNICODE[4002] := 16#8BA5;
   // GBK_TO_UNICODE[4003] := 16#5AE2;
   // GBK_TO_UNICODE[4004] := 16#8BA6;
   // GBK_TO_UNICODE[4005] := 16#5AE4;
   // GBK_TO_UNICODE[4006] := 16#8BA7;
   // GBK_TO_UNICODE[4007] := 16#5AE5;
   // GBK_TO_UNICODE[4008] := 16#8BA8;
   // GBK_TO_UNICODE[4009] := 16#5AE7;
   // GBK_TO_UNICODE[4010] := 16#8BA9;
   // GBK_TO_UNICODE[4011] := 16#5AE8;
   // GBK_TO_UNICODE[4012] := 16#8BAA;
   // GBK_TO_UNICODE[4013] := 16#5AEA;
   // GBK_TO_UNICODE[4014] := 16#8BAB;
   // GBK_TO_UNICODE[4015] := 16#5AEC;
   // GBK_TO_UNICODE[4016] := 16#8BAC;
   // GBK_TO_UNICODE[4017] := 16#5AED;
   // GBK_TO_UNICODE[4018] := 16#8BAD;
   // GBK_TO_UNICODE[4019] := 16#5AEE;
   // GBK_TO_UNICODE[4020] := 16#8BAE;
   // GBK_TO_UNICODE[4021] := 16#5AEF;
   // GBK_TO_UNICODE[4022] := 16#8BAF;
   // GBK_TO_UNICODE[4023] := 16#5AF0;
   // GBK_TO_UNICODE[4024] := 16#8BB0;
   // GBK_TO_UNICODE[4025] := 16#5AF2;
   // GBK_TO_UNICODE[4026] := 16#8BB1;
   // GBK_TO_UNICODE[4027] := 16#5AF3;
   // GBK_TO_UNICODE[4028] := 16#8BB2;
   // GBK_TO_UNICODE[4029] := 16#5AF4;
   // GBK_TO_UNICODE[4030] := 16#8BB3;
   // GBK_TO_UNICODE[4031] := 16#5AF5;
   // GBK_TO_UNICODE[4032] := 16#8BB4;
   // GBK_TO_UNICODE[4033] := 16#5AF6;
   // GBK_TO_UNICODE[4034] := 16#8BB5;
   // GBK_TO_UNICODE[4035] := 16#5AF7;
   // GBK_TO_UNICODE[4036] := 16#8BB6;
   // GBK_TO_UNICODE[4037] := 16#5AF8;
   // GBK_TO_UNICODE[4038] := 16#8BB7;
   // GBK_TO_UNICODE[4039] := 16#5AF9;
   // GBK_TO_UNICODE[4040] := 16#8BB8;
   // GBK_TO_UNICODE[4041] := 16#5AFA;
   // GBK_TO_UNICODE[4042] := 16#8BB9;
   // GBK_TO_UNICODE[4043] := 16#5AFB;
   // GBK_TO_UNICODE[4044] := 16#8BBA;
   // GBK_TO_UNICODE[4045] := 16#5AFC;
   // GBK_TO_UNICODE[4046] := 16#8BBB;
   // GBK_TO_UNICODE[4047] := 16#5AFD;
   // GBK_TO_UNICODE[4048] := 16#8BBC;
   // GBK_TO_UNICODE[4049] := 16#5AFE;
   // GBK_TO_UNICODE[4050] := 16#8BBD;
   // GBK_TO_UNICODE[4051] := 16#5AFF;
   // GBK_TO_UNICODE[4052] := 16#8BBE;
   // GBK_TO_UNICODE[4053] := 16#5B00;
   // GBK_TO_UNICODE[4054] := 16#8BBF;
   // GBK_TO_UNICODE[4055] := 16#5B01;
   // GBK_TO_UNICODE[4056] := 16#8BC0;
   // GBK_TO_UNICODE[4057] := 16#5B02;
   // GBK_TO_UNICODE[4058] := 16#8BC1;
   // GBK_TO_UNICODE[4059] := 16#5B03;
   // GBK_TO_UNICODE[4060] := 16#8BC2;
   // GBK_TO_UNICODE[4061] := 16#5B04;
   // GBK_TO_UNICODE[4062] := 16#8BC3;
   // GBK_TO_UNICODE[4063] := 16#5B05;
   // GBK_TO_UNICODE[4064] := 16#8BC4;
   // GBK_TO_UNICODE[4065] := 16#5B06;
   // GBK_TO_UNICODE[4066] := 16#8BC5;
   // GBK_TO_UNICODE[4067] := 16#5B07;
   // GBK_TO_UNICODE[4068] := 16#8BC6;
   // GBK_TO_UNICODE[4069] := 16#5B08;
   // GBK_TO_UNICODE[4070] := 16#8BC7;
   // GBK_TO_UNICODE[4071] := 16#5B0A;
   // GBK_TO_UNICODE[4072] := 16#8BC8;
   // GBK_TO_UNICODE[4073] := 16#5B0B;
   // GBK_TO_UNICODE[4074] := 16#8BC9;
   // GBK_TO_UNICODE[4075] := 16#5B0C;
   // GBK_TO_UNICODE[4076] := 16#8BCA;
   // GBK_TO_UNICODE[4077] := 16#5B0D;
   // GBK_TO_UNICODE[4078] := 16#8BCB;
   // GBK_TO_UNICODE[4079] := 16#5B0E;
   // GBK_TO_UNICODE[4080] := 16#8BCC;
   // GBK_TO_UNICODE[4081] := 16#5B0F;
   // GBK_TO_UNICODE[4082] := 16#8BCD;
   // GBK_TO_UNICODE[4083] := 16#5B10;
   // GBK_TO_UNICODE[4084] := 16#8BCE;
   // GBK_TO_UNICODE[4085] := 16#5B11;
   // GBK_TO_UNICODE[4086] := 16#8BCF;
   // GBK_TO_UNICODE[4087] := 16#5B12;
   // GBK_TO_UNICODE[4088] := 16#8BD0;
   // GBK_TO_UNICODE[4089] := 16#5B13;
   // GBK_TO_UNICODE[4090] := 16#8BD1;
   // GBK_TO_UNICODE[4091] := 16#5B14;
   // GBK_TO_UNICODE[4092] := 16#8BD2;
   // GBK_TO_UNICODE[4093] := 16#5B15;
   // GBK_TO_UNICODE[4094] := 16#8BD3;
   // GBK_TO_UNICODE[4095] := 16#5B18;
   // GBK_TO_UNICODE[4096] := 16#8BD4;
   // GBK_TO_UNICODE[4097] := 16#5B19;
   // GBK_TO_UNICODE[4098] := 16#8BD5;
   // GBK_TO_UNICODE[4099] := 16#5B1A;
   // GBK_TO_UNICODE[4100] := 16#8BD6;
   // GBK_TO_UNICODE[4101] := 16#5B1B;
   // GBK_TO_UNICODE[4102] := 16#8BD7;
   // GBK_TO_UNICODE[4103] := 16#5B1C;
   // GBK_TO_UNICODE[4104] := 16#8BD8;
   // GBK_TO_UNICODE[4105] := 16#5B1D;
   // GBK_TO_UNICODE[4106] := 16#8BD9;
   // GBK_TO_UNICODE[4107] := 16#5B1E;
   // GBK_TO_UNICODE[4108] := 16#8BDA;
   // GBK_TO_UNICODE[4109] := 16#5B1F;
   // GBK_TO_UNICODE[4110] := 16#8BDB;
   // GBK_TO_UNICODE[4111] := 16#5B20;
   // GBK_TO_UNICODE[4112] := 16#8BDC;
   // GBK_TO_UNICODE[4113] := 16#5B21;
   // GBK_TO_UNICODE[4114] := 16#8BDD;
   // GBK_TO_UNICODE[4115] := 16#5B22;
   // GBK_TO_UNICODE[4116] := 16#8BDE;
   // GBK_TO_UNICODE[4117] := 16#5B23;
   // GBK_TO_UNICODE[4118] := 16#8BDF;
   // GBK_TO_UNICODE[4119] := 16#5B24;
   // GBK_TO_UNICODE[4120] := 16#8BE0;
   // GBK_TO_UNICODE[4121] := 16#5B25;
   // GBK_TO_UNICODE[4122] := 16#8BE1;
   // GBK_TO_UNICODE[4123] := 16#5B26;
   // GBK_TO_UNICODE[4124] := 16#8BE2;
   // GBK_TO_UNICODE[4125] := 16#5B27;
   // GBK_TO_UNICODE[4126] := 16#8BE3;
   // GBK_TO_UNICODE[4127] := 16#5B28;
   // GBK_TO_UNICODE[4128] := 16#8BE4;
   // GBK_TO_UNICODE[4129] := 16#5B29;
   // GBK_TO_UNICODE[4130] := 16#8BE5;
   // GBK_TO_UNICODE[4131] := 16#5B2A;
   // GBK_TO_UNICODE[4132] := 16#8BE6;
   // GBK_TO_UNICODE[4133] := 16#5B2B;
   // GBK_TO_UNICODE[4134] := 16#8BE7;
   // GBK_TO_UNICODE[4135] := 16#5B2C;
   // GBK_TO_UNICODE[4136] := 16#8BE8;
   // GBK_TO_UNICODE[4137] := 16#5B2D;
   // GBK_TO_UNICODE[4138] := 16#8BE9;
   // GBK_TO_UNICODE[4139] := 16#5B2E;
   // GBK_TO_UNICODE[4140] := 16#8BEA;
   // GBK_TO_UNICODE[4141] := 16#5B2F;
   // GBK_TO_UNICODE[4142] := 16#8BEB;
   // GBK_TO_UNICODE[4143] := 16#5B30;
   // GBK_TO_UNICODE[4144] := 16#8BEC;
   // GBK_TO_UNICODE[4145] := 16#5B31;
   // GBK_TO_UNICODE[4146] := 16#8BED;
   // GBK_TO_UNICODE[4147] := 16#5B33;
   // GBK_TO_UNICODE[4148] := 16#8BEE;
   // GBK_TO_UNICODE[4149] := 16#5B35;
   // GBK_TO_UNICODE[4150] := 16#8BEF;
   // GBK_TO_UNICODE[4151] := 16#5B36;
   // GBK_TO_UNICODE[4152] := 16#8BF0;
   // GBK_TO_UNICODE[4153] := 16#5B38;
   // GBK_TO_UNICODE[4154] := 16#8BF1;
   // GBK_TO_UNICODE[4155] := 16#5B39;
   // GBK_TO_UNICODE[4156] := 16#8BF2;
   // GBK_TO_UNICODE[4157] := 16#5B3A;
   // GBK_TO_UNICODE[4158] := 16#8BF3;
   // GBK_TO_UNICODE[4159] := 16#5B3B;
   // GBK_TO_UNICODE[4160] := 16#8BF4;
   // GBK_TO_UNICODE[4161] := 16#5B3C;
   // GBK_TO_UNICODE[4162] := 16#8BF5;
   // GBK_TO_UNICODE[4163] := 16#5B3D;
   // GBK_TO_UNICODE[4164] := 16#8BF6;
   // GBK_TO_UNICODE[4165] := 16#5B3E;
   // GBK_TO_UNICODE[4166] := 16#8BF7;
   // GBK_TO_UNICODE[4167] := 16#5B3F;
   // GBK_TO_UNICODE[4168] := 16#8BF8;
   // GBK_TO_UNICODE[4169] := 16#5B41;
   // GBK_TO_UNICODE[4170] := 16#8BF9;
   // GBK_TO_UNICODE[4171] := 16#5B42;
   // GBK_TO_UNICODE[4172] := 16#8BFA;
   // GBK_TO_UNICODE[4173] := 16#5B43;
   // GBK_TO_UNICODE[4174] := 16#8BFB;
   // GBK_TO_UNICODE[4175] := 16#5B44;
   // GBK_TO_UNICODE[4176] := 16#8BFC;
   // GBK_TO_UNICODE[4177] := 16#5B45;
   // GBK_TO_UNICODE[4178] := 16#8BFD;
   // GBK_TO_UNICODE[4179] := 16#5B46;
   // GBK_TO_UNICODE[4180] := 16#8BFE;
   // GBK_TO_UNICODE[4181] := 16#5B47;
   // GBK_TO_UNICODE[4182] := 16#8C40;
   // GBK_TO_UNICODE[4183] := 16#5B48;
   // GBK_TO_UNICODE[4184] := 16#8C41;
   // GBK_TO_UNICODE[4185] := 16#5B49;
   // GBK_TO_UNICODE[4186] := 16#8C42;
   // GBK_TO_UNICODE[4187] := 16#5B4A;
   // GBK_TO_UNICODE[4188] := 16#8C43;
   // GBK_TO_UNICODE[4189] := 16#5B4B;
   // GBK_TO_UNICODE[4190] := 16#8C44;
   // GBK_TO_UNICODE[4191] := 16#5B4C;
   // GBK_TO_UNICODE[4192] := 16#8C45;
   // GBK_TO_UNICODE[4193] := 16#5B4D;
   // GBK_TO_UNICODE[4194] := 16#8C46;
   // GBK_TO_UNICODE[4195] := 16#5B4E;
   // GBK_TO_UNICODE[4196] := 16#8C47;
   // GBK_TO_UNICODE[4197] := 16#5B4F;
   // GBK_TO_UNICODE[4198] := 16#8C48;
   // GBK_TO_UNICODE[4199] := 16#5B52;
   // GBK_TO_UNICODE[4200] := 16#8C49;
   // GBK_TO_UNICODE[4201] := 16#5B56;
   // GBK_TO_UNICODE[4202] := 16#8C4A;
   // GBK_TO_UNICODE[4203] := 16#5B5E;
   // GBK_TO_UNICODE[4204] := 16#8C4B;
   // GBK_TO_UNICODE[4205] := 16#5B60;
   // GBK_TO_UNICODE[4206] := 16#8C4C;
   // GBK_TO_UNICODE[4207] := 16#5B61;
   // GBK_TO_UNICODE[4208] := 16#8C4D;
   // GBK_TO_UNICODE[4209] := 16#5B67;
   // GBK_TO_UNICODE[4210] := 16#8C4E;
   // GBK_TO_UNICODE[4211] := 16#5B68;
   // GBK_TO_UNICODE[4212] := 16#8C4F;
   // GBK_TO_UNICODE[4213] := 16#5B6B;
   // GBK_TO_UNICODE[4214] := 16#8C50;
   // GBK_TO_UNICODE[4215] := 16#5B6D;
   // GBK_TO_UNICODE[4216] := 16#8C51;
   // GBK_TO_UNICODE[4217] := 16#5B6E;
   // GBK_TO_UNICODE[4218] := 16#8C52;
   // GBK_TO_UNICODE[4219] := 16#5B6F;
   // GBK_TO_UNICODE[4220] := 16#8C53;
   // GBK_TO_UNICODE[4221] := 16#5B72;
   // GBK_TO_UNICODE[4222] := 16#8C54;
   // GBK_TO_UNICODE[4223] := 16#5B74;
   // GBK_TO_UNICODE[4224] := 16#8C55;
   // GBK_TO_UNICODE[4225] := 16#5B76;
   // GBK_TO_UNICODE[4226] := 16#8C56;
   // GBK_TO_UNICODE[4227] := 16#5B77;
   // GBK_TO_UNICODE[4228] := 16#8C57;
   // GBK_TO_UNICODE[4229] := 16#5B78;
   // GBK_TO_UNICODE[4230] := 16#8C58;
   // GBK_TO_UNICODE[4231] := 16#5B79;
   // GBK_TO_UNICODE[4232] := 16#8C59;
   // GBK_TO_UNICODE[4233] := 16#5B7B;
   // GBK_TO_UNICODE[4234] := 16#8C5A;
   // GBK_TO_UNICODE[4235] := 16#5B7C;
   // GBK_TO_UNICODE[4236] := 16#8C5B;
   // GBK_TO_UNICODE[4237] := 16#5B7E;
   // GBK_TO_UNICODE[4238] := 16#8C5C;
   // GBK_TO_UNICODE[4239] := 16#5B7F;
   // GBK_TO_UNICODE[4240] := 16#8C5D;
   // GBK_TO_UNICODE[4241] := 16#5B82;
   // GBK_TO_UNICODE[4242] := 16#8C5E;
   // GBK_TO_UNICODE[4243] := 16#5B86;
   // GBK_TO_UNICODE[4244] := 16#8C5F;
   // GBK_TO_UNICODE[4245] := 16#5B8A;
   // GBK_TO_UNICODE[4246] := 16#8C60;
   // GBK_TO_UNICODE[4247] := 16#5B8D;
   // GBK_TO_UNICODE[4248] := 16#8C61;
   // GBK_TO_UNICODE[4249] := 16#5B8E;
   // GBK_TO_UNICODE[4250] := 16#8C62;
   // GBK_TO_UNICODE[4251] := 16#5B90;
   // GBK_TO_UNICODE[4252] := 16#8C63;
   // GBK_TO_UNICODE[4253] := 16#5B91;
   // GBK_TO_UNICODE[4254] := 16#8C64;
   // GBK_TO_UNICODE[4255] := 16#5B92;
   // GBK_TO_UNICODE[4256] := 16#8C65;
   // GBK_TO_UNICODE[4257] := 16#5B94;
   // GBK_TO_UNICODE[4258] := 16#8C66;
   // GBK_TO_UNICODE[4259] := 16#5B96;
   // GBK_TO_UNICODE[4260] := 16#8C67;
   // GBK_TO_UNICODE[4261] := 16#5B9F;
   // GBK_TO_UNICODE[4262] := 16#8C68;
   // GBK_TO_UNICODE[4263] := 16#5BA7;
   // GBK_TO_UNICODE[4264] := 16#8C69;
   // GBK_TO_UNICODE[4265] := 16#5BA8;
   // GBK_TO_UNICODE[4266] := 16#8C6A;
   // GBK_TO_UNICODE[4267] := 16#5BA9;
   // GBK_TO_UNICODE[4268] := 16#8C6B;
   // GBK_TO_UNICODE[4269] := 16#5BAC;
   // GBK_TO_UNICODE[4270] := 16#8C6C;
   // GBK_TO_UNICODE[4271] := 16#5BAD;
   // GBK_TO_UNICODE[4272] := 16#8C6D;
   // GBK_TO_UNICODE[4273] := 16#5BAE;
   // GBK_TO_UNICODE[4274] := 16#8C6E;
   // GBK_TO_UNICODE[4275] := 16#5BAF;
   // GBK_TO_UNICODE[4276] := 16#8C6F;
   // GBK_TO_UNICODE[4277] := 16#5BB1;
   // GBK_TO_UNICODE[4278] := 16#8C70;
   // GBK_TO_UNICODE[4279] := 16#5BB2;
   // GBK_TO_UNICODE[4280] := 16#8C71;
   // GBK_TO_UNICODE[4281] := 16#5BB7;
   // GBK_TO_UNICODE[4282] := 16#8C72;
   // GBK_TO_UNICODE[4283] := 16#5BBA;
   // GBK_TO_UNICODE[4284] := 16#8C73;
   // GBK_TO_UNICODE[4285] := 16#5BBB;
   // GBK_TO_UNICODE[4286] := 16#8C74;
   // GBK_TO_UNICODE[4287] := 16#5BBC;
   // GBK_TO_UNICODE[4288] := 16#8C75;
   // GBK_TO_UNICODE[4289] := 16#5BC0;
   // GBK_TO_UNICODE[4290] := 16#8C76;
   // GBK_TO_UNICODE[4291] := 16#5BC1;
   // GBK_TO_UNICODE[4292] := 16#8C77;
   // GBK_TO_UNICODE[4293] := 16#5BC3;
   // GBK_TO_UNICODE[4294] := 16#8C78;
   // GBK_TO_UNICODE[4295] := 16#5BC8;
   // GBK_TO_UNICODE[4296] := 16#8C79;
   // GBK_TO_UNICODE[4297] := 16#5BC9;
   // GBK_TO_UNICODE[4298] := 16#8C7A;
   // GBK_TO_UNICODE[4299] := 16#5BCA;
   // GBK_TO_UNICODE[4300] := 16#8C7B;
   // GBK_TO_UNICODE[4301] := 16#5BCB;
   // GBK_TO_UNICODE[4302] := 16#8C7C;
   // GBK_TO_UNICODE[4303] := 16#5BCD;
   // GBK_TO_UNICODE[4304] := 16#8C7D;
   // GBK_TO_UNICODE[4305] := 16#5BCE;
   // GBK_TO_UNICODE[4306] := 16#8C7E;
   // GBK_TO_UNICODE[4307] := 16#5BCF;
   // GBK_TO_UNICODE[4308] := 16#8C80;
   // GBK_TO_UNICODE[4309] := 16#5BD1;
   // GBK_TO_UNICODE[4310] := 16#8C81;
   // GBK_TO_UNICODE[4311] := 16#5BD4;
   // GBK_TO_UNICODE[4312] := 16#8C82;
   // GBK_TO_UNICODE[4313] := 16#5BD5;
   // GBK_TO_UNICODE[4314] := 16#8C83;
   // GBK_TO_UNICODE[4315] := 16#5BD6;
   // GBK_TO_UNICODE[4316] := 16#8C84;
   // GBK_TO_UNICODE[4317] := 16#5BD7;
   // GBK_TO_UNICODE[4318] := 16#8C85;
   // GBK_TO_UNICODE[4319] := 16#5BD8;
   // GBK_TO_UNICODE[4320] := 16#8C86;
   // GBK_TO_UNICODE[4321] := 16#5BD9;
   // GBK_TO_UNICODE[4322] := 16#8C87;
   // GBK_TO_UNICODE[4323] := 16#5BDA;
   // GBK_TO_UNICODE[4324] := 16#8C88;
   // GBK_TO_UNICODE[4325] := 16#5BDB;
   // GBK_TO_UNICODE[4326] := 16#8C89;
   // GBK_TO_UNICODE[4327] := 16#5BDC;
   // GBK_TO_UNICODE[4328] := 16#8C8A;
   // GBK_TO_UNICODE[4329] := 16#5BE0;
   // GBK_TO_UNICODE[4330] := 16#8C8B;
   // GBK_TO_UNICODE[4331] := 16#5BE2;
   // GBK_TO_UNICODE[4332] := 16#8C8C;
   // GBK_TO_UNICODE[4333] := 16#5BE3;
   // GBK_TO_UNICODE[4334] := 16#8C8D;
   // GBK_TO_UNICODE[4335] := 16#5BE6;
   // GBK_TO_UNICODE[4336] := 16#8C8E;
   // GBK_TO_UNICODE[4337] := 16#5BE7;
   // GBK_TO_UNICODE[4338] := 16#8C8F;
   // GBK_TO_UNICODE[4339] := 16#5BE9;
   // GBK_TO_UNICODE[4340] := 16#8C90;
   // GBK_TO_UNICODE[4341] := 16#5BEA;
   // GBK_TO_UNICODE[4342] := 16#8C91;
   // GBK_TO_UNICODE[4343] := 16#5BEB;
   // GBK_TO_UNICODE[4344] := 16#8C92;
   // GBK_TO_UNICODE[4345] := 16#5BEC;
   // GBK_TO_UNICODE[4346] := 16#8C93;
   // GBK_TO_UNICODE[4347] := 16#5BED;
   // GBK_TO_UNICODE[4348] := 16#8C94;
   // GBK_TO_UNICODE[4349] := 16#5BEF;
   // GBK_TO_UNICODE[4350] := 16#8C95;
   // GBK_TO_UNICODE[4351] := 16#5BF1;
   // GBK_TO_UNICODE[4352] := 16#8C96;
   // GBK_TO_UNICODE[4353] := 16#5BF2;
   // GBK_TO_UNICODE[4354] := 16#8C97;
   // GBK_TO_UNICODE[4355] := 16#5BF3;
   // GBK_TO_UNICODE[4356] := 16#8C98;
   // GBK_TO_UNICODE[4357] := 16#5BF4;
   // GBK_TO_UNICODE[4358] := 16#8C99;
   // GBK_TO_UNICODE[4359] := 16#5BF5;
   // GBK_TO_UNICODE[4360] := 16#8C9A;
   // GBK_TO_UNICODE[4361] := 16#5BF6;
   // GBK_TO_UNICODE[4362] := 16#8C9B;
   // GBK_TO_UNICODE[4363] := 16#5BF7;
   // GBK_TO_UNICODE[4364] := 16#8C9C;
   // GBK_TO_UNICODE[4365] := 16#5BFD;
   // GBK_TO_UNICODE[4366] := 16#8C9D;
   // GBK_TO_UNICODE[4367] := 16#5BFE;
   // GBK_TO_UNICODE[4368] := 16#8C9E;
   // GBK_TO_UNICODE[4369] := 16#5C00;
   // GBK_TO_UNICODE[4370] := 16#8C9F;
   // GBK_TO_UNICODE[4371] := 16#5C02;
   // GBK_TO_UNICODE[4372] := 16#8CA0;
   // GBK_TO_UNICODE[4373] := 16#5C03;
   // GBK_TO_UNICODE[4374] := 16#8CA1;
   // GBK_TO_UNICODE[4375] := 16#5C05;
   // GBK_TO_UNICODE[4376] := 16#8CA2;
   // GBK_TO_UNICODE[4377] := 16#5C07;
   // GBK_TO_UNICODE[4378] := 16#8CA3;
   // GBK_TO_UNICODE[4379] := 16#5C08;
   // GBK_TO_UNICODE[4380] := 16#8CA4;
   // GBK_TO_UNICODE[4381] := 16#5C0B;
   // GBK_TO_UNICODE[4382] := 16#8CA5;
   // GBK_TO_UNICODE[4383] := 16#5C0C;
   // GBK_TO_UNICODE[4384] := 16#8CA6;
   // GBK_TO_UNICODE[4385] := 16#5C0D;
   // GBK_TO_UNICODE[4386] := 16#8CA7;
   // GBK_TO_UNICODE[4387] := 16#5C0E;
   // GBK_TO_UNICODE[4388] := 16#8CA8;
   // GBK_TO_UNICODE[4389] := 16#5C10;
   // GBK_TO_UNICODE[4390] := 16#8CA9;
   // GBK_TO_UNICODE[4391] := 16#5C12;
   // GBK_TO_UNICODE[4392] := 16#8CAA;
   // GBK_TO_UNICODE[4393] := 16#5C13;
   // GBK_TO_UNICODE[4394] := 16#8CAB;
   // GBK_TO_UNICODE[4395] := 16#5C17;
   // GBK_TO_UNICODE[4396] := 16#8CAC;
   // GBK_TO_UNICODE[4397] := 16#5C19;
   // GBK_TO_UNICODE[4398] := 16#8CAD;
   // GBK_TO_UNICODE[4399] := 16#5C1B;
   // GBK_TO_UNICODE[4400] := 16#8CAE;
   // GBK_TO_UNICODE[4401] := 16#5C1E;
   // GBK_TO_UNICODE[4402] := 16#8CAF;
   // GBK_TO_UNICODE[4403] := 16#5C1F;
   // GBK_TO_UNICODE[4404] := 16#8CB0;
   // GBK_TO_UNICODE[4405] := 16#5C20;
   // GBK_TO_UNICODE[4406] := 16#8CB1;
   // GBK_TO_UNICODE[4407] := 16#5C21;
   // GBK_TO_UNICODE[4408] := 16#8CB2;
   // GBK_TO_UNICODE[4409] := 16#5C23;
   // GBK_TO_UNICODE[4410] := 16#8CB3;
   // GBK_TO_UNICODE[4411] := 16#5C26;
   // GBK_TO_UNICODE[4412] := 16#8CB4;
   // GBK_TO_UNICODE[4413] := 16#5C28;
   // GBK_TO_UNICODE[4414] := 16#8CB5;
   // GBK_TO_UNICODE[4415] := 16#5C29;
   // GBK_TO_UNICODE[4416] := 16#8CB6;
   // GBK_TO_UNICODE[4417] := 16#5C2A;
   // GBK_TO_UNICODE[4418] := 16#8CB7;
   // GBK_TO_UNICODE[4419] := 16#5C2B;
   // GBK_TO_UNICODE[4420] := 16#8CB8;
   // GBK_TO_UNICODE[4421] := 16#5C2D;
   // GBK_TO_UNICODE[4422] := 16#8CB9;
   // GBK_TO_UNICODE[4423] := 16#5C2E;
   // GBK_TO_UNICODE[4424] := 16#8CBA;
   // GBK_TO_UNICODE[4425] := 16#5C2F;
   // GBK_TO_UNICODE[4426] := 16#8CBB;
   // GBK_TO_UNICODE[4427] := 16#5C30;
   // GBK_TO_UNICODE[4428] := 16#8CBC;
